C07272=1088.539,208.717,-73.617,176.065,20.904,153.231
C07273=1088.530,208.334,-73.580,176.061,20.901,153.231
C07274=1088.507,207.310,-73.481,175.988,20.864,153.235
C07275=1088.502,207.061,-73.457,175.986,20.863,153.235
C07276=1088.497,206.812,-73.433,175.983,20.861,153.235
C07277=1088.490,206.563,-73.409,175.980,20.859,153.235
C07278=1088.485,206.314,-73.385,175.977,20.858,153.236
C07279=1088.479,206.066,-73.361,175.974,20.857,153.236
C07280=1088.474,205.817,-73.337,175.972,20.855,153.236
C07281=1088.469,205.568,-73.314,175.969,20.854,153.236
C07282=1088.463,205.320,-73.290,175.965,20.852,153.236
C07283=1088.457,205.071,-73.265,175.963,20.851,153.236
C07284=1088.452,204.821,-73.242,175.960,20.850,153.237
C07285=1088.446,204.573,-73.218,175.958,20.848,153.237
C07286=1088.441,204.324,-73.195,175.955,20.847,153.237
C07287=1088.435,204.076,-73.171,175.952,20.845,153.237
C07288=1088.429,203.827,-73.147,175.949,20.844,153.237
C07289=1088.424,203.578,-73.123,175.946,20.842,153.237
C07290=1088.418,203.329,-73.099,175.944,20.841,153.237
C07291=1088.413,203.080,-73.076,175.941,20.839,153.237
C07292=1088.407,202.831,-73.052,175.938,20.838,153.238
C07293=1088.402,202.582,-73.028,175.936,20.837,153.238
C07294=1088.396,202.334,-73.005,175.933,20.836,153.238
C07295=1088.391,202.085,-72.981,175.929,20.834,153.238
C07296=1088.385,201.836,-72.957,175.927,20.833,153.238
C07297=1088.378,201.587,-72.934,175.924,20.831,153.238
C07298=1088.373,201.338,-72.910,175.922,20.830,153.239
C07299=1088.367,201.089,-72.887,175.919,20.829,153.239
C07300=1088.361,200.841,-72.863,175.916,20.827,153.239
C07301=1088.356,200.592,-72.840,175.914,20.826,153.239
C07302=1088.350,200.344,-72.816,175.910,20.824,153.239
C07303=1088.345,200.095,-72.793,175.907,20.823,153.239
C07304=1088.340,199.845,-72.770,175.905,20.822,153.240
C07305=1088.334,199.597,-72.746,175.902,20.820,153.240
C07306=1088.327,199.348,-72.723,175.899,20.819,153.240
C07307=1088.322,199.098,-72.699,175.897,20.818,153.240
C07308=1088.316,198.850,-72.675,175.894,20.816,153.240
C07309=1088.310,198.601,-72.652,175.891,20.814,153.240
C07310=1088.305,198.353,-72.628,175.888,20.813,153.241
C07311=1088.299,198.104,-72.605,175.885,20.812,153.241
C07312=1088.294,197.855,-72.582,175.883,20.811,153.241
C07313=1088.289,197.606,-72.559,175.880,20.809,153.241
C07314=1088.283,197.357,-72.535,175.877,20.808,153.241
C07315=1088.277,197.108,-72.512,175.875,20.807,153.241
C07316=1088.272,196.859,-72.489,175.872,20.805,153.241
C07317=1088.266,196.611,-72.465,175.870,20.804,153.241
C07318=1088.260,196.362,-72.442,175.866,20.802,153.242
C07319=1088.254,196.113,-72.419,175.863,20.801,153.242
C07320=1088.249,195.864,-72.396,175.861,20.800,153.242
C07321=1088.244,195.615,-72.373,175.858,20.798,153.242
C07322=1088.238,195.367,-72.349,175.856,20.797,153.242
C07323=1088.233,195.118,-72.325,175.853,20.795,153.242
C07324=1088.227,194.869,-72.302,175.850,20.794,153.243
C07325=1088.221,194.620,-72.279,175.848,20.793,153.243
C07326=1088.216,194.371,-72.257,175.845,20.791,153.243
C07327=1088.211,194.122,-72.233,175.842,20.790,153.243
C07328=1088.205,193.873,-72.209,175.840,20.788,153.243
C07329=1088.199,193.624,-72.186,175.836,20.787,153.243
C07330=1088.193,193.376,-72.163,175.834,20.786,153.243
C07331=1088.187,193.127,-72.141,175.831,20.784,153.244
C07332=1088.182,192.877,-72.117,175.828,20.783,153.244
C07333=1088.177,192.629,-72.094,175.826,20.781,153.244
C07334=1088.171,192.380,-72.071,175.823,20.780,153.244
C07335=1088.165,192.103,-72.046,175.821,20.778,153.244
C07336=1088.159,191.825,-72.019,175.817,20.777,153.244
C07337=1088.153,191.548,-71.994,175.814,20.775,153.244
C07338=1088.146,191.270,-71.968,175.811,20.774,153.245
C07339=1088.141,191.021,-71.945,175.808,20.772,153.245
C07340=1088.135,190.772,-71.922,175.806,20.771,153.245
C07341=1088.130,190.523,-71.899,175.803,20.769,153.245
C07342=1088.125,190.275,-71.876,175.801,20.768,153.245
C07343=1088.119,190.026,-71.853,175.798,20.766,153.245
C07344=1088.113,189.777,-71.831,175.795,20.765,153.245
C07345=1088.108,189.528,-71.807,175.793,20.763,153.245
C07346=1088.102,189.279,-71.784,175.790,20.762,153.246
C07347=1088.097,189.030,-71.761,175.787,20.761,153.246
C07348=1088.091,188.782,-71.739,175.785,20.760,153.246
C07349=1088.086,188.533,-71.716,175.782,20.758,153.246
C07350=1088.080,188.284,-71.693,175.780,20.757,153.246
C07351=1088.075,188.035,-71.670,175.777,20.755,153.246
C07352=1088.070,187.786,-71.647,175.775,20.754,153.246
C07353=1088.064,187.537,-71.624,175.771,20.752,153.246
C07354=1088.059,187.289,-71.601,175.768,20.750,153.247
C07355=1088.053,187.040,-71.578,175.766,20.749,153.247
C07356=1088.048,186.790,-71.556,175.763,20.748,153.247
C07357=1088.042,186.541,-71.533,175.761,20.746,153.247
C07358=1088.037,186.293,-71.511,175.758,20.745,153.247
C07359=1088.031,186.044,-71.488,175.756,20.743,153.247
C07360=1088.025,185.795,-71.465,175.753,20.742,153.247
C07361=1088.021,185.545,-71.442,175.750,20.740,153.247
C07362=1088.015,185.297,-71.419,175.748,20.739,153.247
C07363=1088.010,185.048,-71.396,175.745,20.737,153.248
C07364=1088.003,184.800,-71.374,175.743,20.736,153.248
C07365=1087.998,184.550,-71.352,175.740,20.735,153.248
C07366=1087.992,184.301,-71.329,175.737,20.734,153.248
C07367=1087.986,184.053,-71.306,175.735,20.732,153.248
C07368=1087.981,183.803,-71.284,175.732,20.731,153.248
C07369=1087.974,183.554,-71.261,175.729,20.729,153.248
C07370=1087.969,183.306,-71.239,175.727,20.728,153.249
C07371=1087.964,183.057,-71.217,175.724,20.727,153.249
C07372=1087.958,182.808,-71.194,175.722,20.725,153.249
C07373=1087.952,182.559,-71.171,175.719,20.724,153.249
C07374=1087.946,182.310,-71.149,175.716,20.722,153.249
C07375=1087.941,182.061,-71.126,175.714,20.722,153.249
C07376=1087.935,181.813,-71.104,175.711,20.720,153.249
C07377=1087.929,181.563,-71.082,175.708,20.719,153.250
C07378=1087.924,181.315,-71.059,175.706,20.717,153.250
C07379=1087.918,181.065,-71.037,175.703,20.716,153.250
C07380=1087.912,180.816,-71.014,175.701,20.714,153.250
C07381=1087.907,180.568,-70.992,175.698,20.713,153.250
C07382=1087.901,180.319,-70.969,175.695,20.712,153.250
C07383=1087.895,180.070,-70.947,175.693,20.710,153.250
C07384=1087.889,179.821,-70.925,175.690,20.709,153.251
C07385=1087.884,179.572,-70.902,175.687,20.708,153.251
C07386=1087.878,179.323,-70.881,175.685,20.706,153.251
C07387=1087.872,179.074,-70.858,175.682,20.705,153.251
C07388=1087.867,178.825,-70.836,175.680,20.703,153.251
C07389=1087.861,178.576,-70.814,175.677,20.702,153.251
C07390=1087.855,178.327,-70.791,175.675,20.700,153.251
C07391=1087.850,178.078,-70.769,175.672,20.699,153.252
C07392=1087.844,177.829,-70.747,175.669,20.698,153.252
C07393=1087.839,177.580,-70.725,175.667,20.696,153.252
C07394=1087.833,177.332,-70.702,175.664,20.695,153.252
C07395=1087.827,177.082,-70.680,175.661,20.694,153.252
C07396=1087.822,176.834,-70.658,175.659,20.692,153.252
C07397=1087.816,176.585,-70.635,175.656,20.691,153.252
C07398=1087.810,176.335,-70.614,175.654,20.689,153.252
C07399=1087.804,176.058,-70.589,175.651,20.688,153.252
C07400=1087.798,175.780,-70.564,175.648,20.686,153.253
C07401=1087.792,175.502,-70.539,175.645,20.684,153.253
C07402=1087.785,175.225,-70.515,175.642,20.683,153.253
C07403=1087.780,174.976,-70.493,175.640,20.682,153.253
C07404=1087.774,174.727,-70.471,175.637,20.680,153.253
C07405=1087.768,174.477,-70.449,175.635,20.679,153.253
C07406=1087.763,174.229,-70.426,175.632,20.677,153.253
C07407=1087.757,173.980,-70.405,175.630,20.676,153.253
C07408=1087.752,173.731,-70.383,175.627,20.674,153.254
C07409=1087.746,173.482,-70.361,175.624,20.673,153.254
C07410=1087.740,173.233,-70.338,175.623,20.672,153.254
C07411=1087.736,172.984,-70.316,175.620,20.670,153.254
C07412=1087.729,172.735,-70.295,175.617,20.669,153.254
C07413=1087.724,172.486,-70.272,175.615,20.668,153.254
C07414=1087.718,172.238,-70.250,175.612,20.666,153.254
C07415=1087.713,171.988,-70.228,175.610,20.665,153.254
C07416=1087.707,171.740,-70.207,175.607,20.663,153.254
C07417=1087.702,171.490,-70.185,175.605,20.662,153.255
C07418=1087.696,171.242,-70.163,175.602,20.660,153.255
C07419=1087.691,170.992,-70.141,175.600,20.658,153.255
C07420=1087.685,170.743,-70.119,175.597,20.657,153.255
C07421=1087.679,170.495,-70.097,175.594,20.655,153.255
C07422=1087.674,170.245,-70.075,175.592,20.654,153.255
C07423=1087.668,169.997,-70.053,175.589,20.653,153.255
C07424=1087.663,169.747,-70.031,175.587,20.651,153.255
C07425=1087.657,169.499,-70.010,175.584,20.650,153.255
C07426=1087.652,169.249,-69.988,175.582,20.649,153.255
C07427=1087.646,169.001,-69.966,175.580,20.647,153.256
C07428=1087.641,168.751,-69.944,175.577,20.645,153.256
C07429=1087.635,168.503,-69.923,175.575,20.644,153.256
C07430=1087.630,168.253,-69.901,175.572,20.642,153.256
C07431=1087.624,168.005,-69.879,175.570,20.641,153.256
C07432=1087.619,167.755,-69.857,175.567,20.640,153.256
C07433=1087.613,167.507,-69.836,175.564,20.638,153.256
C07434=1087.608,167.257,-69.814,175.562,20.637,153.256
C07435=1087.603,167.009,-69.792,175.560,20.635,153.256
C07436=1087.597,166.759,-69.770,175.557,20.633,153.256
C07437=1087.592,166.511,-69.749,175.554,20.632,153.257
C07438=1087.587,166.262,-69.727,175.553,20.631,153.257
C07439=1087.581,166.012,-69.705,175.550,20.629,153.257
C07440=1087.575,165.764,-69.684,175.548,20.627,153.257
C07441=1087.570,165.514,-69.662,175.545,20.626,153.257
C07442=1087.564,165.266,-69.641,175.543,20.625,153.257
C07443=1087.559,165.016,-69.618,175.540,20.623,153.257
C07444=1087.553,164.767,-69.598,175.537,20.622,153.257
C07445=1087.548,164.519,-69.576,175.535,20.620,153.257
C07446=1087.542,164.269,-69.554,175.532,20.618,153.257
C07447=1087.537,164.021,-69.533,175.530,20.617,153.257
C07448=1087.531,163.771,-69.511,175.528,20.616,153.257
C07449=1087.526,163.523,-69.490,175.526,20.614,153.257
C07450=1087.521,163.274,-69.468,175.523,20.613,153.258
C07451=1087.515,163.024,-69.447,175.521,20.611,153.258
C07452=1087.510,162.775,-69.425,175.518,20.610,153.258
C07453=1087.505,162.527,-69.404,175.516,20.608,153.258
C07454=1087.499,162.278,-69.382,175.513,20.606,153.258
C07455=1087.494,162.028,-69.361,175.510,20.605,153.258
C07456=1087.488,161.779,-69.339,175.509,20.603,153.258
C07457=1087.482,161.530,-69.318,175.506,20.602,153.258
C07458=1087.477,161.282,-69.296,175.504,20.600,153.258
C07459=1087.472,161.032,-69.275,175.501,20.599,153.258
C07460=1087.466,160.783,-69.254,175.499,20.598,153.258
C07461=1087.460,160.534,-69.232,175.496,20.596,153.258
C07462=1087.454,160.286,-69.211,175.494,20.594,153.259
C07463=1087.449,160.007,-69.187,175.491,20.593,153.259
C07464=1087.442,159.729,-69.164,175.489,20.591,153.259
C07465=1087.436,159.451,-69.140,175.486,20.590,153.259
C07466=1087.429,159.173,-69.117,175.483,20.588,153.259
C07467=1087.424,158.924,-69.095,175.481,20.586,153.259
C07468=1087.419,158.675,-69.074,175.478,20.585,153.259
C07469=1087.413,158.425,-69.052,175.476,20.584,153.259
C07470=1087.407,158.177,-69.031,175.473,20.582,153.259
C07471=1087.402,157.928,-69.011,175.471,20.580,153.259
C07472=1087.396,157.679,-68.989,175.468,20.579,153.260
C07473=1087.390,157.430,-68.968,175.467,20.578,153.260
C07474=1087.385,157.181,-68.947,175.464,20.576,153.260
C07475=1087.379,156.932,-68.926,175.461,20.575,153.260
C07476=1087.374,156.683,-68.905,175.459,20.573,153.260
C07477=1087.368,156.434,-68.884,175.456,20.571,153.260
C07478=1087.363,156.184,-68.862,175.454,20.570,153.260
C07479=1087.357,155.936,-68.841,175.452,20.568,153.260
C07480=1087.352,155.686,-68.820,175.450,20.567,153.260
C07481=1087.346,155.437,-68.799,175.447,20.566,153.260
C07482=1087.341,155.188,-68.778,175.445,20.564,153.260
C07483=1087.335,154.940,-68.757,175.442,20.562,153.260
C07484=1087.329,154.690,-68.736,175.440,20.561,153.260
C07485=1087.324,154.441,-68.715,175.437,20.559,153.261
C07486=1087.318,154.192,-68.694,175.435,20.558,153.261
C07487=1087.312,153.943,-68.673,175.433,20.556,153.261
C07488=1087.306,153.694,-68.653,175.430,20.555,153.261
C07489=1087.301,153.445,-68.632,175.428,20.554,153.261
C07490=1087.295,153.196,-68.610,175.425,20.552,153.261
C07491=1087.290,152.947,-68.590,175.423,20.550,153.261
C07492=1087.284,152.698,-68.569,175.421,20.549,153.261
C07493=1087.279,152.449,-68.548,175.419,20.548,153.261
C07494=1087.273,152.199,-68.527,175.416,20.546,153.261
C07495=1087.267,151.951,-68.506,175.414,20.544,153.261
C07496=1087.262,151.702,-68.485,175.411,20.543,153.261
C07497=1087.257,151.452,-68.465,175.410,20.541,153.261
C07498=1087.251,151.203,-68.443,175.407,20.540,153.262
C07499=1087.245,150.954,-68.423,175.404,20.539,153.262
C07500=1087.240,150.705,-68.402,175.402,20.537,153.262
C07501=1087.235,150.456,-68.381,175.399,20.535,153.262
C07502=1087.228,150.207,-68.360,175.397,20.534,153.262
C07503=1087.223,149.958,-68.340,175.395,20.532,153.262
C07504=1087.217,149.709,-68.319,175.393,20.531,153.262
C07505=1087.212,149.460,-68.298,175.390,20.529,153.262
C07506=1087.206,149.210,-68.277,175.388,20.527,153.262
C07507=1087.201,148.961,-68.257,175.385,20.526,153.262
C07508=1087.195,148.713,-68.235,175.384,20.525,153.262
C07509=1087.189,148.464,-68.215,175.381,20.523,153.262
C07510=1087.184,148.215,-68.195,175.379,20.522,153.262
C07511=1087.178,147.965,-68.174,175.376,20.520,153.262
C07512=1087.173,147.716,-68.153,175.374,20.518,153.262
C07513=1087.167,147.468,-68.133,175.372,20.517,153.263
C07514=1087.161,147.219,-68.112,175.369,20.516,153.263
C07515=1087.156,146.969,-68.091,175.367,20.514,153.263
C07516=1087.150,146.720,-68.071,175.364,20.512,153.263
C07517=1087.144,146.471,-68.051,175.362,20.511,153.263
C07518=1087.139,146.222,-68.030,175.360,20.509,153.263
C07519=1087.134,145.973,-68.010,175.358,20.508,153.263
C07520=1087.127,145.724,-67.989,175.355,20.506,153.263
C07521=1087.122,145.475,-67.968,175.353,20.505,153.263
C07522=1087.116,145.225,-67.947,175.351,20.504,153.263
C07523=1087.111,144.976,-67.927,175.349,20.502,153.263
C07524=1087.105,144.727,-67.907,175.346,20.500,153.263
C07525=1087.100,144.478,-67.886,175.344,20.498,153.263
C07526=1087.094,144.229,-67.865,175.341,20.497,153.263
C07527=1087.087,143.951,-67.843,175.339,20.495,153.264
C07528=1087.081,143.672,-67.820,175.336,20.493,153.264
C07529=1087.075,143.394,-67.797,175.334,20.492,153.264
C07530=1087.069,143.116,-67.774,175.331,20.490,153.264
C07531=1087.064,142.867,-67.754,175.329,20.489,153.264
C07532=1087.057,142.618,-67.733,175.327,20.487,153.264
C07533=1087.052,142.368,-67.714,175.325,20.486,153.264
C07534=1087.047,142.119,-67.693,175.322,20.484,153.264
C07535=1087.041,141.870,-67.673,175.320,20.482,153.264
C07536=1087.036,141.621,-67.652,175.317,20.480,153.264
C07537=1087.030,141.372,-67.632,175.316,20.479,153.264
C07538=1087.025,141.123,-67.612,175.313,20.477,153.264
C07539=1087.019,140.874,-67.591,175.311,20.476,153.264
C07540=1087.013,140.625,-67.571,175.308,20.474,153.264
C07541=1087.008,140.376,-67.551,175.307,20.473,153.264
C07542=1087.001,140.126,-67.531,175.304,20.471,153.264
C07543=1086.996,139.877,-67.510,175.302,20.470,153.264
C07544=1086.990,139.628,-67.490,175.299,20.468,153.264
C07545=1086.985,139.379,-67.470,175.298,20.467,153.264
C07546=1086.980,139.129,-67.450,175.295,20.465,153.264
C07547=1086.974,138.881,-67.430,175.293,20.463,153.264
C07548=1086.969,138.632,-67.409,175.290,20.461,153.264
C07549=1086.963,138.383,-67.389,175.289,20.460,153.265
C07550=1086.957,138.134,-67.369,175.286,20.459,153.265
C07551=1086.952,137.884,-67.349,175.284,20.457,153.265
C07552=1086.946,137.635,-67.329,175.281,20.455,153.265
C07553=1086.941,137.386,-67.309,175.280,20.454,153.265
C07554=1086.935,137.137,-67.289,175.277,20.452,153.265
C07555=1086.929,136.888,-67.268,175.275,20.451,153.265
C07556=1086.924,136.639,-67.249,175.272,20.449,153.265
C07557=1086.918,136.389,-67.228,175.271,20.448,153.265
C07558=1086.912,136.140,-67.208,175.268,20.446,153.265
C07559=1086.906,135.891,-67.188,175.266,20.444,153.265
C07560=1086.901,135.642,-67.168,175.264,20.443,153.265
C07561=1086.895,135.393,-67.148,175.262,20.442,153.265
C07562=1086.890,135.144,-67.128,175.259,20.440,153.265
C07563=1086.884,134.894,-67.109,175.257,20.438,153.265
C07564=1086.879,134.645,-67.088,175.255,20.437,153.265
C07565=1086.873,134.396,-67.068,175.253,20.435,153.265
C07566=1086.867,134.147,-67.049,175.250,20.433,153.265
C07567=1086.862,133.898,-67.028,175.248,20.431,153.265
C07568=1086.856,133.649,-67.008,175.246,20.430,153.265
C07569=1086.851,133.399,-66.989,175.244,20.428,153.265
C07570=1086.845,133.150,-66.969,175.241,20.427,153.265
C07571=1086.839,132.902,-66.949,175.240,20.425,153.265
C07572=1086.834,132.653,-66.929,175.237,20.424,153.265
C07573=1086.828,132.404,-66.909,175.235,20.422,153.266
C07574=1086.823,132.154,-66.890,175.232,20.420,153.266
C07575=1086.817,131.905,-66.869,175.231,20.419,153.266
C07576=1086.811,131.656,-66.849,175.228,20.417,153.266
C07577=1086.806,131.407,-66.830,175.226,20.416,153.266
C07578=1086.800,131.158,-66.810,175.224,20.414,153.266
C07579=1086.794,130.909,-66.791,175.222,20.412,153.266
C07580=1086.789,130.660,-66.770,175.219,20.411,153.266
C07581=1086.783,130.410,-66.751,175.217,20.409,153.266
C07582=1086.777,130.161,-66.731,175.215,20.408,153.266
C07583=1086.771,129.912,-66.712,175.213,20.406,153.266
C07584=1086.765,129.663,-66.692,175.210,20.405,153.266
C07585=1086.760,129.414,-66.673,175.209,20.403,153.266
C07586=1086.755,129.165,-66.652,175.206,20.401,153.266
C07587=1086.749,128.915,-66.633,175.204,20.400,153.266
C07588=1086.743,128.666,-66.613,175.202,20.398,153.266
C07589=1086.737,128.417,-66.594,175.200,20.397,153.266
C07590=1086.731,128.167,-66.575,175.197,20.395,153.266
C07591=1086.725,127.889,-66.553,175.195,20.393,153.266
C07592=1086.719,127.611,-66.530,175.192,20.391,153.266
C07593=1086.713,127.332,-66.509,175.190,20.389,153.266
C07594=1086.706,127.054,-66.487,175.188,20.388,153.266
C07595=1086.700,126.805,-66.467,175.185,20.386,153.266
C07596=1086.694,126.556,-66.448,175.184,20.385,153.266
C07597=1086.689,126.306,-66.428,175.181,20.383,153.266
C07598=1086.683,126.057,-66.408,175.179,20.381,153.266
C07599=1086.678,125.808,-66.388,175.177,20.380,153.266
C07600=1086.673,125.559,-66.370,175.175,20.378,153.266
C07601=1086.667,125.310,-66.350,175.172,20.376,153.266
C07602=1086.661,125.061,-66.330,175.171,20.375,153.266
C07603=1086.655,124.811,-66.311,175.168,20.373,153.266
C07604=1086.649,124.563,-66.291,175.166,20.371,153.267
C07605=1086.644,124.313,-66.272,175.164,20.370,153.266
C07606=1086.638,124.064,-66.253,175.162,20.368,153.266
C07607=1086.633,123.815,-66.234,175.160,20.366,153.266
C07608=1086.627,123.566,-66.214,175.158,20.365,153.267
C07609=1086.621,123.317,-66.195,175.156,20.363,153.267
C07610=1086.615,123.067,-66.175,175.153,20.361,153.267
C07611=1086.610,122.818,-66.156,175.152,20.360,153.266
C07612=1086.604,122.569,-66.136,175.149,20.358,153.267
C07613=1086.599,122.320,-66.117,175.147,20.356,153.267
C07614=1086.594,122.071,-66.097,175.145,20.355,153.267
C07615=1086.588,121.821,-66.078,175.143,20.353,153.267
C07616=1086.582,121.572,-66.059,175.140,20.351,153.267
C07617=1086.576,121.323,-66.039,175.139,20.350,153.267
C07618=1086.571,121.074,-66.020,175.137,20.348,153.267
C07619=1086.566,120.825,-66.001,175.134,20.346,153.267
C07620=1086.560,120.575,-65.982,175.133,20.345,153.267
C07621=1086.554,120.326,-65.962,175.130,20.343,153.267
C07622=1086.548,120.076,-65.943,175.128,20.341,153.267
C07623=1086.543,119.828,-65.924,175.126,20.340,153.267
C07624=1086.537,119.579,-65.904,175.124,20.338,153.267
C07625=1086.532,119.329,-65.885,175.122,20.336,153.267
C07626=1086.526,119.080,-65.866,175.120,20.334,153.267
C07627=1086.521,118.831,-65.847,175.118,20.333,153.267
C07628=1086.515,118.582,-65.828,175.115,20.331,153.267
C07629=1086.510,118.332,-65.808,175.114,20.329,153.267
C07630=1086.504,118.084,-65.790,175.111,20.327,153.267
C07631=1086.499,117.834,-65.770,175.109,20.326,153.267
C07632=1086.493,117.585,-65.751,175.107,20.324,153.267
C07633=1086.487,117.335,-65.732,175.105,20.322,153.267
C07634=1086.482,117.087,-65.713,175.103,20.321,153.267
C07635=1086.477,116.837,-65.694,175.101,20.319,153.267
C07636=1086.471,116.588,-65.675,175.099,20.317,153.267
C07637=1086.466,116.339,-65.656,175.097,20.316,153.267
C07638=1086.460,116.090,-65.636,175.095,20.314,153.267
C07639=1086.454,115.840,-65.617,175.092,20.312,153.267
C07640=1086.449,115.592,-65.599,175.091,20.310,153.266
C07641=1086.443,115.342,-65.580,175.089,20.308,153.266
C07642=1086.437,115.093,-65.560,175.086,20.306,153.266
C07643=1086.432,114.844,-65.541,175.085,20.305,153.266
C07644=1086.427,114.595,-65.522,175.082,20.303,153.266
C07645=1086.421,114.345,-65.503,175.080,20.301,153.266
C07646=1086.416,114.097,-65.484,175.079,20.300,153.266
C07647=1086.410,113.846,-65.466,175.076,20.298,153.266
C07648=1086.404,113.597,-65.447,175.075,20.297,153.266
C07649=1086.398,113.348,-65.428,175.072,20.295,153.266
C07650=1086.393,113.099,-65.409,175.070,20.293,153.266
C07651=1086.387,112.850,-65.390,175.068,20.291,153.266
C07652=1086.381,112.601,-65.371,175.066,20.289,153.266
C07653=1086.376,112.352,-65.352,175.064,20.287,153.266
C07654=1086.371,112.102,-65.334,175.062,20.286,153.266
C07655=1086.364,111.824,-65.312,175.060,20.284,153.266
C07656=1086.358,111.545,-65.291,175.057,20.282,153.266
C07657=1086.351,111.267,-65.270,175.055,20.280,153.266
C07658=1086.345,110.988,-65.249,175.053,20.278,153.266
C07659=1086.340,110.739,-65.231,175.050,20.276,153.266
C07660=1086.334,110.490,-65.212,175.049,20.275,153.266
C07661=1086.328,110.241,-65.193,175.046,20.273,153.266
C07662=1086.322,109.992,-65.174,175.045,20.272,153.266
C07663=1086.317,109.742,-65.156,175.042,20.270,153.266
C07664=1086.311,109.493,-65.137,175.040,20.268,153.266
C07665=1086.305,109.244,-65.118,175.039,20.266,153.266
C07666=1086.300,108.995,-65.099,175.036,20.264,153.266
C07667=1086.294,108.745,-65.081,175.035,20.263,153.266
C07668=1086.288,108.496,-65.062,175.032,20.261,153.266
C07669=1086.283,108.247,-65.043,175.030,20.259,153.266
C07670=1086.277,107.998,-65.025,175.029,20.257,153.266
C07671=1086.271,107.748,-65.006,175.026,20.256,153.266
C07672=1086.266,107.499,-64.987,175.025,20.254,153.266
C07673=1086.260,107.250,-64.969,175.022,20.252,153.266
C07674=1086.255,107.001,-64.950,175.020,20.251,153.266
C07675=1086.248,106.751,-64.931,175.018,20.249,153.266
C07676=1086.243,106.502,-64.913,175.016,20.247,153.266
C07677=1086.237,106.253,-64.895,175.014,20.246,153.266
C07678=1086.232,106.004,-64.876,175.012,20.244,153.266
C07679=1086.226,105.754,-64.857,175.010,20.242,153.266
C07680=1086.221,105.506,-64.839,175.008,20.240,153.266
C07681=1086.215,105.256,-64.820,175.006,20.238,153.266
C07682=1086.209,105.007,-64.802,175.005,20.236,153.266
C07683=1086.204,104.757,-64.784,175.002,20.234,153.266
C07684=1086.198,104.508,-64.765,175.000,20.232,153.266
C07685=1086.193,104.259,-64.746,174.998,20.231,153.266
C07686=1086.186,104.010,-64.728,174.996,20.229,153.266
C07687=1086.181,103.761,-64.709,174.995,20.228,153.266
C07688=1086.176,103.511,-64.691,174.992,20.226,153.266
C07689=1086.170,103.262,-64.672,174.990,20.224,153.266
C07690=1086.165,103.012,-64.654,174.988,20.222,153.266
C07691=1086.159,102.764,-64.636,174.986,20.220,153.266
C07692=1086.154,102.514,-64.617,174.985,20.219,153.266
C07693=1086.148,102.265,-64.599,174.982,20.217,153.266
C07694=1086.142,102.015,-64.580,174.981,20.215,153.266
C07695=1086.136,101.767,-64.562,174.978,20.213,153.266
C07696=1086.131,101.517,-64.544,174.976,20.211,153.266
C07697=1086.126,101.268,-64.526,174.975,20.209,153.265
C07698=1086.120,101.018,-64.507,174.972,20.207,153.265
C07699=1086.114,100.769,-64.489,174.971,20.206,153.265
C07700=1086.108,100.520,-64.471,174.969,20.204,153.265
C07701=1086.103,100.270,-64.452,174.966,20.202,153.265
C07702=1086.097,100.021,-64.434,174.965,20.201,153.265
C07703=1086.091,99.772,-64.416,174.962,20.199,153.265
C07704=1086.086,99.523,-64.398,174.961,20.197,153.265
C07705=1086.079,99.274,-64.379,174.959,20.195,153.265
C07706=1086.074,99.025,-64.361,174.957,20.194,153.265
C07707=1086.069,98.775,-64.343,174.955,20.192,153.265
C07708=1086.063,98.526,-64.325,174.953,20.190,153.265
C07709=1086.057,98.276,-64.307,174.951,20.188,153.265
C07710=1086.052,98.027,-64.288,174.949,20.186,153.265
C07711=1086.045,97.778,-64.270,174.947,20.185,153.265
C07712=1086.040,97.529,-64.252,174.945,20.183,153.265
C07713=1086.034,97.280,-64.235,174.943,20.181,153.265
C07714=1086.029,97.030,-64.215,174.941,20.179,153.265
C07715=1086.023,96.781,-64.198,174.940,20.177,153.265
C07716=1086.017,96.532,-64.180,174.937,20.175,153.265
C07717=1086.012,96.282,-64.162,174.935,20.173,153.265
C07718=1086.006,96.033,-64.143,174.933,20.172,153.265
C07719=1086.000,95.755,-64.124,174.931,20.170,153.265
C07720=1085.993,95.477,-64.104,174.929,20.168,153.265
C07721=1085.987,95.198,-64.082,174.927,20.166,153.265
C07722=1085.981,94.919,-64.063,174.925,20.164,153.264
C07723=1085.975,94.671,-64.045,174.923,20.162,153.264
C07724=1085.969,94.421,-64.027,174.921,20.160,153.264
C07725=1085.964,94.172,-64.009,174.919,20.158,153.264
C07726=1085.958,93.922,-63.991,174.917,20.156,153.264
C07727=1085.953,93.673,-63.973,174.915,20.155,153.264
C07728=1085.947,93.425,-63.955,174.913,20.153,153.264
C07729=1085.941,93.175,-63.936,174.912,20.151,153.264
C07730=1085.936,92.925,-63.919,174.909,20.149,153.264
C07731=1085.930,92.676,-63.901,174.908,20.147,153.264
C07732=1085.924,92.427,-63.883,174.906,20.145,153.264
C07733=1085.919,92.177,-63.865,174.903,20.143,153.264
C07734=1085.913,91.928,-63.847,174.902,20.141,153.264
C07735=1085.908,91.679,-63.830,174.900,20.139,153.264
C07736=1085.902,91.430,-63.812,174.898,20.138,153.264
C07737=1085.896,91.180,-63.793,174.896,20.136,153.264
C07738=1085.891,90.931,-63.775,174.895,20.134,153.264
C07739=1085.886,90.682,-63.758,174.892,20.132,153.264
C07740=1085.879,90.432,-63.740,174.891,20.131,153.263
C07741=1085.874,90.183,-63.722,174.888,20.129,153.263
C07742=1085.868,89.933,-63.704,174.887,20.127,153.263
C07743=1085.862,89.684,-63.687,174.885,20.125,153.263
C07744=1085.857,89.435,-63.669,174.883,20.123,153.263
C07745=1085.851,89.186,-63.651,174.881,20.121,153.263
C07746=1085.845,88.937,-63.634,174.879,20.120,153.263
C07747=1085.839,88.687,-63.616,174.877,20.118,153.263
C07748=1085.834,88.438,-63.598,174.875,20.116,153.263
C07749=1085.828,88.189,-63.581,174.873,20.114,153.263
C07750=1085.822,87.939,-63.563,174.871,20.112,153.263
C07751=1085.816,87.690,-63.545,174.870,20.110,153.263
C07752=1085.811,87.441,-63.528,174.867,20.108,153.263
C07753=1085.805,87.191,-63.510,174.866,20.106,153.263
C07754=1085.799,86.942,-63.492,174.864,20.104,153.263
C07755=1085.794,86.693,-63.474,174.862,20.103,153.263
C07756=1085.788,86.443,-63.457,174.860,20.101,153.263
C07757=1085.782,86.194,-63.440,174.859,20.099,153.262
C07758=1085.777,85.945,-63.422,174.856,20.097,153.262
C07759=1085.771,85.695,-63.404,174.855,20.096,153.262
C07760=1085.765,85.446,-63.387,174.852,20.094,153.262
C07761=1085.760,85.197,-63.369,174.851,20.092,153.262
C07762=1085.754,84.948,-63.351,174.849,20.090,153.262
C07763=1085.748,84.698,-63.334,174.847,20.088,153.262
C07764=1085.743,84.449,-63.316,174.845,20.086,153.262
C07765=1085.737,84.199,-63.299,174.844,20.084,153.262
C07766=1085.731,83.950,-63.281,174.841,20.082,153.262
C07767=1085.726,83.701,-63.264,174.840,20.081,153.262
C07768=1085.720,83.452,-63.246,174.838,20.078,153.262
C07769=1085.715,83.203,-63.228,174.836,20.077,153.262
C07770=1085.708,82.952,-63.212,174.834,20.075,153.262
C07771=1085.703,82.703,-63.194,174.833,20.073,153.262
C07772=1085.697,82.454,-63.177,174.830,20.071,153.262
C07773=1085.692,82.205,-63.159,174.829,20.069,153.262
C07774=1085.685,81.956,-63.141,174.827,20.067,153.261
C07775=1085.680,81.706,-63.124,174.825,20.065,153.261
C07776=1085.675,81.457,-63.107,174.823,20.063,153.261
C07777=1085.669,81.208,-63.089,174.822,20.061,153.261
C07778=1085.664,80.959,-63.072,174.819,20.060,153.261
C07779=1085.658,80.708,-63.054,174.818,20.058,153.261
C07780=1085.652,80.459,-63.037,174.816,20.056,153.261
C07781=1085.647,80.210,-63.019,174.814,20.054,153.261
C07782=1085.641,79.961,-63.003,174.812,20.052,153.261
C07783=1085.635,79.683,-62.984,174.810,20.050,153.261
C07784=1085.628,79.405,-62.963,174.808,20.047,153.261
C07785=1085.622,79.126,-62.944,174.806,20.046,153.261
C07786=1085.615,78.848,-62.925,174.804,20.043,153.260
C07787=1085.610,78.598,-62.908,174.802,20.041,153.260
C07788=1085.605,78.349,-62.891,174.801,20.039,153.260
C07789=1085.599,78.099,-62.873,174.798,20.037,153.260
C07790=1085.593,77.850,-62.856,174.797,20.036,153.260
C07791=1085.587,77.601,-62.839,174.795,20.033,153.260
C07792=1085.582,77.352,-62.822,174.793,20.032,153.260
C07793=1085.576,77.102,-62.805,174.791,20.030,153.260
C07794=1085.570,76.853,-62.787,174.790,20.028,153.260
C07795=1085.564,76.603,-62.770,174.787,20.026,153.260
C07796=1085.559,76.354,-62.753,174.786,20.024,153.260
C07797=1085.554,76.105,-62.736,174.784,20.022,153.260
C07798=1085.547,75.856,-62.719,174.782,20.020,153.260
C07799=1085.541,75.606,-62.701,174.781,20.018,153.259
C07800=1085.536,75.356,-62.684,174.779,20.016,153.259
C07801=1085.530,75.108,-62.667,174.777,20.015,153.259
C07802=1085.525,74.858,-62.650,174.775,20.012,153.259
C07803=1085.519,74.609,-62.633,174.773,20.011,153.259
C07804=1085.513,74.360,-62.617,174.771,20.009,153.259
C07805=1085.507,74.110,-62.599,174.770,20.007,153.259
C07806=1085.502,73.860,-62.582,174.767,20.005,153.259
C07807=1085.495,73.612,-62.565,174.766,20.003,153.259
C07808=1085.490,73.362,-62.548,174.764,20.001,153.259
C07809=1085.485,73.113,-62.530,174.763,19.999,153.259
C07810=1085.479,72.864,-62.514,174.760,19.997,153.259
C07811=1085.474,72.614,-62.497,174.759,19.995,153.258
C07812=1085.468,72.365,-62.480,174.757,19.993,153.258
C07813=1085.462,72.115,-62.464,174.755,19.992,153.258
C07814=1085.456,71.866,-62.446,174.753,19.989,153.258
C07815=1085.451,71.616,-62.429,174.752,19.988,153.258
C07816=1085.445,71.367,-62.412,174.750,19.985,153.258
C07817=1085.439,71.118,-62.395,174.748,19.984,153.258
C07818=1085.433,70.868,-62.379,174.747,19.982,153.258
C07819=1085.428,70.619,-62.361,174.744,19.980,153.258
C07820=1085.423,70.370,-62.344,174.743,19.978,153.258
C07821=1085.417,70.120,-62.328,174.741,19.976,153.258
C07822=1085.411,69.871,-62.310,174.740,19.974,153.257
C07823=1085.405,69.622,-62.294,174.737,19.972,153.257
C07824=1085.400,69.372,-62.277,174.736,19.970,153.257
C07825=1085.393,69.123,-62.260,174.734,19.968,153.257
C07826=1085.388,68.873,-62.243,174.732,19.966,153.257
C07827=1085.382,68.624,-62.227,174.730,19.964,153.257
C07828=1085.376,68.375,-62.209,174.729,19.962,153.257
C07829=1085.371,68.125,-62.193,174.727,19.960,153.257
C07830=1085.365,67.876,-62.176,174.725,19.958,153.257
C07831=1085.359,67.627,-62.159,174.724,19.956,153.257
C07832=1085.354,67.377,-62.142,174.721,19.954,153.257
C07833=1085.348,67.128,-62.126,174.720,19.952,153.256
C07834=1085.343,66.878,-62.109,174.718,19.950,153.256
C07835=1085.336,66.630,-62.092,174.717,19.948,153.256
C07836=1085.331,66.380,-62.075,174.714,19.946,153.256
C07837=1085.325,66.131,-62.059,174.713,19.944,153.256
C07838=1085.320,65.881,-62.042,174.711,19.943,153.256
C07839=1085.314,65.632,-62.026,174.709,19.941,153.256
C07840=1085.309,65.383,-62.009,174.708,19.939,153.256
C07841=1085.303,65.133,-61.992,174.706,19.937,153.256
C07842=1085.297,64.884,-61.976,174.704,19.935,153.256
C07843=1085.291,64.634,-61.959,174.702,19.933,153.255
C07844=1085.286,64.385,-61.943,174.701,19.931,153.255
C07845=1085.279,64.135,-61.926,174.699,19.929,153.255
C07846=1085.273,63.886,-61.909,174.697,19.927,153.255
C07847=1085.268,63.608,-61.891,174.695,19.925,153.255
C07848=1085.261,63.329,-61.872,174.693,19.923,153.255
C07849=1085.254,63.051,-61.854,174.691,19.921,153.255
C07850=1085.247,62.772,-61.835,174.689,19.919,153.255
C07851=1085.241,62.523,-61.819,174.688,19.917,153.255
C07852=1085.235,62.274,-61.803,174.686,19.915,153.255
C07853=1085.230,62.024,-61.786,174.684,19.913,153.255
C07854=1085.224,61.775,-61.770,174.682,19.911,153.255
C07855=1085.218,61.525,-61.753,174.681,19.909,153.254
C07856=1085.212,61.276,-61.737,174.678,19.907,153.254
C07857=1085.207,61.026,-61.720,174.677,19.905,153.254
C07858=1085.201,60.777,-61.704,174.676,19.903,153.254
C07859=1085.195,60.528,-61.688,174.674,19.901,153.254
C07860=1085.189,60.278,-61.671,174.672,19.899,153.254
C07861=1085.183,60.029,-61.655,174.670,19.897,153.254
C07862=1085.178,59.779,-61.638,174.669,19.895,153.254
C07863=1085.172,59.531,-61.621,174.666,19.893,153.254
C07864=1085.166,59.281,-61.605,174.665,19.891,153.254
C07865=1085.160,59.031,-61.590,174.664,19.889,153.253
C07866=1085.154,58.782,-61.573,174.661,19.887,153.253
C07867=1085.149,58.532,-61.556,174.660,19.885,153.253
C07868=1085.143,58.283,-61.540,174.658,19.883,153.253
C07869=1085.137,58.034,-61.524,174.657,19.881,153.253
C07870=1085.131,57.784,-61.508,174.654,19.879,153.253
C07871=1085.125,57.535,-61.491,174.653,19.877,153.253
C07872=1085.119,57.286,-61.475,174.651,19.876,153.253
C07873=1085.114,57.036,-61.458,174.649,19.873,153.253
C07874=1085.108,56.786,-61.442,174.648,19.871,153.252
C07875=1085.102,56.537,-61.426,174.646,19.869,153.252
C07876=1085.097,56.289,-61.410,174.645,19.867,153.252
C07877=1085.091,56.039,-61.394,174.642,19.865,153.252
C07878=1085.085,55.790,-61.377,174.641,19.863,153.252
C07879=1085.080,55.540,-61.361,174.639,19.862,153.252
C07880=1085.074,55.290,-61.345,174.637,19.859,153.252
C07881=1085.068,55.041,-61.329,174.636,19.857,153.252
C07882=1085.062,54.791,-61.313,174.634,19.855,153.252
C07883=1085.056,54.542,-61.296,174.633,19.853,153.252
C07884=1085.050,54.293,-61.280,174.631,19.852,153.252
C07885=1085.044,54.043,-61.264,174.629,19.849,153.251
C07886=1085.040,53.794,-61.248,174.628,19.847,153.251
C07887=1085.034,53.545,-61.232,174.625,19.845,153.251
C07888=1085.028,53.295,-61.215,174.624,19.843,153.251
C07889=1085.022,53.046,-61.199,174.623,19.842,153.251
C07890=1085.016,52.796,-61.183,174.621,19.839,153.251
C07891=1085.011,52.546,-61.167,174.619,19.837,153.251
C07892=1085.005,52.297,-61.151,174.617,19.835,153.251
C07893=1084.999,52.049,-61.135,174.616,19.833,153.250
C07894=1084.993,51.799,-61.119,174.614,19.831,153.250
C07895=1084.988,51.549,-61.103,174.612,19.829,153.250
C07896=1084.983,51.300,-61.087,174.611,19.827,153.250
C07897=1084.977,51.050,-61.070,174.609,19.825,153.250
C07898=1084.971,50.802,-61.054,174.607,19.823,153.250
C07899=1084.966,50.552,-61.039,174.605,19.821,153.250
C07900=1084.960,50.302,-61.023,174.604,19.819,153.250
C07901=1084.954,50.053,-61.006,174.603,19.818,153.250
C07902=1084.948,49.803,-60.991,174.600,19.815,153.249
C07903=1084.943,49.554,-60.975,174.599,19.813,153.249
C07904=1084.937,49.305,-60.959,174.597,19.811,153.249
C07905=1084.931,49.055,-60.943,174.596,19.809,153.249
C07906=1084.925,48.806,-60.927,174.594,19.807,153.249
C07907=1084.919,48.556,-60.911,174.592,19.805,153.249
C07908=1084.914,48.307,-60.895,174.591,19.803,153.249
C07909=1084.908,48.058,-60.879,174.589,19.801,153.249
C07910=1084.903,47.808,-60.862,174.587,19.799,153.249
C07911=1084.897,47.530,-60.846,174.585,19.797,153.248
C07912=1084.890,47.251,-60.828,174.584,19.795,153.248
C07913=1084.884,46.972,-60.810,174.582,19.792,153.248
C07914=1084.878,46.694,-60.792,174.580,19.790,153.248
C07915=1084.872,46.444,-60.776,174.578,19.788,153.248
C07916=1084.866,46.194,-60.760,174.577,19.786,153.248
C07917=1084.861,45.945,-60.745,174.575,19.784,153.248
C07918=1084.855,45.696,-60.729,174.574,19.782,153.247
C07919=1084.849,45.446,-60.712,174.572,19.779,153.247
C07920=1084.844,45.196,-60.697,174.570,19.778,153.247
C07921=1084.838,44.948,-60.681,174.569,19.776,153.247
C07922=1084.833,44.698,-60.666,174.567,19.773,153.247
C07923=1084.827,44.449,-60.649,174.565,19.771,153.247
C07924=1084.822,44.199,-60.634,174.564,19.770,153.247
C07925=1084.816,43.950,-60.618,174.562,19.767,153.246
C07926=1084.810,43.700,-60.602,174.561,19.765,153.246
C07927=1084.804,43.451,-60.586,174.559,19.763,153.246
C07928=1084.799,43.201,-60.571,174.557,19.761,153.246
C07929=1084.793,42.951,-60.555,174.556,19.759,153.246
C07930=1084.787,42.702,-60.540,174.554,19.757,153.246
C07931=1084.782,42.453,-60.524,174.552,19.755,153.246
C07932=1084.776,42.204,-60.508,174.550,19.753,153.246
C07933=1084.770,41.954,-60.493,174.549,19.751,153.245
C07934=1084.764,41.704,-60.476,174.547,19.749,153.245
C07935=1084.758,41.455,-60.462,174.545,19.747,153.245
C07936=1084.752,41.206,-60.446,174.544,19.744,153.245
C07937=1084.747,40.956,-60.430,174.543,19.743,153.245
C07938=1084.742,40.707,-60.415,174.541,19.741,153.245
C07939=1084.736,40.458,-60.399,174.539,19.738,153.245
C07940=1084.729,40.208,-60.384,174.538,19.736,153.245
C07941=1084.724,39.959,-60.368,174.536,19.734,153.245
C07942=1084.718,39.709,-60.352,174.535,19.732,153.244
C07943=1084.713,39.459,-60.337,174.532,19.730,153.244
C07944=1084.708,39.210,-60.322,174.531,19.728,153.244
C07945=1084.701,38.961,-60.306,174.530,19.726,153.244
C07946=1084.695,38.711,-60.290,174.528,19.724,153.244
C07947=1084.690,38.462,-60.275,174.526,19.722,153.244
C07948=1084.684,38.212,-60.259,174.525,19.720,153.244
C07949=1084.678,37.963,-60.244,174.523,19.718,153.243
C07950=1084.673,37.713,-60.229,174.522,19.716,153.243
C07951=1084.667,37.464,-60.213,174.520,19.713,153.243
C07952=1084.661,37.214,-60.198,174.518,19.712,153.243
C07953=1084.655,36.965,-60.182,174.517,19.710,153.243
C07954=1084.650,36.715,-60.167,174.515,19.707,153.243
C07955=1084.643,36.466,-60.151,174.513,19.706,153.243
C07956=1084.638,36.217,-60.136,174.512,19.704,153.243
C07957=1084.632,35.967,-60.120,174.510,19.701,153.242
C07958=1084.626,35.717,-60.106,174.508,19.700,153.242
C07959=1084.621,35.469,-60.090,174.507,19.698,153.242
C07960=1084.614,35.219,-60.075,174.505,19.695,153.242
C07961=1084.609,34.969,-60.059,174.504,19.694,153.242
C07962=1084.604,34.720,-60.044,174.502,19.692,153.242
C07963=1084.597,34.471,-60.028,174.500,19.689,153.242
C07964=1084.591,34.221,-60.013,174.499,19.687,153.242
C07965=1084.586,33.972,-59.998,174.498,19.686,153.241
C07966=1084.580,33.722,-59.983,174.496,19.683,153.241
C07967=1084.574,33.473,-59.968,174.494,19.681,153.241
C07968=1084.568,33.223,-59.953,174.492,19.679,153.241
C07969=1084.563,32.974,-59.936,174.491,19.677,153.241
C07970=1084.557,32.725,-59.922,174.489,19.675,153.241
C07971=1084.551,32.475,-59.906,174.487,19.673,153.241
C07972=1084.545,32.226,-59.892,174.486,19.671,153.241
C07973=1084.540,31.976,-59.876,174.485,19.669,153.240
C07974=1084.533,31.726,-59.861,174.483,19.667,153.240
C07975=1084.528,31.447,-59.844,174.481,19.665,153.240
C07976=1084.521,31.169,-59.827,174.479,19.662,153.240
C07977=1084.514,30.890,-59.810,174.478,19.660,153.240
C07978=1084.508,30.612,-59.793,174.476,19.658,153.240
C07979=1084.502,30.362,-59.778,174.475,19.656,153.239
C07980=1084.497,30.113,-59.763,174.472,19.654,153.239
C07981=1084.491,29.863,-59.748,174.471,19.652,153.239
C07982=1084.486,29.614,-59.733,174.470,19.650,153.239
C07983=1084.479,29.364,-59.718,174.468,19.647,153.239
C07984=1084.474,29.115,-59.703,174.466,19.646,153.239
C07985=1084.468,28.866,-59.687,174.465,19.644,153.239
C07986=1084.462,28.617,-59.672,174.463,19.641,153.239
C07987=1084.456,28.367,-59.657,174.462,19.639,153.238
C07988=1084.450,28.117,-59.641,174.460,19.638,153.238
C07989=1084.445,27.868,-59.627,174.458,19.635,153.238
C07990=1084.439,27.618,-59.613,174.457,19.633,153.238
C07991=1084.434,27.368,-59.597,174.456,19.631,153.238
C07992=1084.427,27.119,-59.582,174.453,19.629,153.238
C07993=1084.422,26.869,-59.567,174.452,19.627,153.238
C07994=1084.416,26.620,-59.552,174.451,19.625,153.238
C07995=1084.410,26.371,-59.538,174.449,19.623,153.238
C07996=1084.404,26.121,-59.522,174.447,19.621,153.237
C07997=1084.399,25.872,-59.508,174.446,19.619,153.237
C07998=1084.393,25.622,-59.492,174.444,19.617,153.237
C07999=1084.387,25.373,-59.478,174.443,19.615,153.237
C08000=1084.381,25.123,-59.463,174.441,19.613,153.237
C08001=1084.376,24.874,-59.447,174.439,19.611,153.237
C08002=1084.369,24.624,-59.432,174.438,19.609,153.236
C08003=1084.364,24.375,-59.419,174.437,19.607,153.236
C08004=1084.358,24.125,-59.403,174.435,19.605,153.236
C08005=1084.352,23.876,-59.388,174.433,19.603,153.236
C08006=1084.346,23.626,-59.374,174.432,19.601,153.236
C08007=1084.341,23.377,-59.358,174.430,19.599,153.236
C08008=1084.335,23.127,-59.343,174.429,19.597,153.236
C08009=1084.329,22.878,-59.329,174.427,19.595,153.236
C08010=1084.323,22.628,-59.314,174.425,19.592,153.235
C08011=1084.318,22.379,-59.299,174.424,19.591,153.235
C08012=1084.311,22.129,-59.284,174.422,19.588,153.235
C08013=1084.305,21.880,-59.270,174.421,19.586,153.235
C08014=1084.300,21.630,-59.254,174.419,19.584,153.235
C08015=1084.294,21.381,-59.240,174.418,19.582,153.235
C08016=1084.288,21.131,-59.226,174.416,19.580,153.235
C08017=1084.283,20.882,-59.210,174.414,19.578,153.235
C08018=1084.277,20.633,-59.196,174.413,19.576,153.234
C08019=1084.271,20.383,-59.182,174.412,19.574,153.234
C08020=1084.265,20.134,-59.167,174.410,19.572,153.234
C08021=1084.260,19.884,-59.151,174.408,19.570,153.234
C08022=1084.254,19.635,-59.137,174.407,19.568,153.234
C08023=1084.248,19.384,-59.123,174.405,19.565,153.234
C08024=1084.242,19.135,-59.108,174.404,19.564,153.234
C08025=1084.236,18.886,-59.093,174.402,19.562,153.233
C08026=1084.231,18.636,-59.079,174.401,19.560,153.233
C08027=1084.225,18.387,-59.064,174.399,19.557,153.233
C08028=1084.219,18.137,-59.049,174.398,19.556,153.233
C08029=1084.213,17.888,-59.035,174.396,19.554,153.233
C08030=1084.207,17.638,-59.020,174.394,19.551,153.233
C08031=1084.202,17.389,-59.005,174.393,19.549,153.233
C08032=1084.196,17.139,-58.991,174.392,19.548,153.233
C08033=1084.190,16.890,-58.976,174.389,19.545,153.232
C08034=1084.184,16.641,-58.962,174.388,19.543,153.232
C08035=1084.178,16.390,-58.947,174.387,19.541,153.232
C08036=1084.172,16.141,-58.933,174.386,19.539,153.232
C08037=1084.167,15.891,-58.917,174.383,19.537,153.232
C08038=1084.161,15.642,-58.904,174.382,19.535,153.232
C08039=1084.154,15.365,-58.887,174.380,19.533,153.232
C08040=1084.148,15.088,-58.872,174.379,19.531,153.231
C08041=1084.142,14.811,-58.855,174.377,19.528,153.231
C08042=1084.135,14.533,-58.840,174.376,19.526,153.231
C08043=1084.130,14.284,-58.825,174.374,19.524,153.231
C08044=1084.123,14.035,-58.810,174.372,19.522,153.231
C08045=1084.118,13.785,-58.796,174.371,19.520,153.231
C08046=1084.111,13.535,-58.781,174.370,19.518,153.231
C08047=1084.106,13.286,-58.767,174.368,19.516,153.230
C08048=1084.100,13.036,-58.752,174.366,19.514,153.230
C08049=1084.094,12.787,-58.739,174.365,19.512,153.230
C08050=1084.088,12.538,-58.724,174.363,19.509,153.230
C08051=1084.082,12.287,-58.710,174.361,19.508,153.230
C08052=1084.076,12.038,-58.695,174.360,19.506,153.230
C08053=1084.071,11.789,-58.681,174.359,19.504,153.230
C08054=1084.065,11.539,-58.666,174.357,19.501,153.230
C08055=1084.059,11.290,-58.653,174.355,19.500,153.229
C08056=1084.053,11.040,-58.638,174.354,19.498,153.229
C08057=1084.047,10.790,-58.624,174.352,19.495,153.229
C08058=1084.041,10.541,-58.609,174.351,19.494,153.229
C08059=1084.035,10.291,-58.595,174.349,19.492,153.229
C08060=1084.029,10.042,-58.582,174.348,19.490,153.229
C08061=1084.023,9.793,-58.567,174.346,19.487,153.229
C08062=1084.017,9.543,-58.553,174.345,19.486,153.229
C08063=1084.011,9.294,-58.538,174.343,19.484,153.228
C08064=1084.006,9.044,-58.524,174.341,19.481,153.228
C08065=1084.000,8.794,-58.509,174.340,19.479,153.228
C08066=1083.994,8.545,-58.496,174.339,19.478,153.228
C08067=1083.989,8.295,-58.482,174.337,19.476,153.228
C08068=1083.982,8.046,-58.467,174.335,19.473,153.228
C08069=1083.977,7.796,-58.453,174.334,19.472,153.228
C08070=1083.971,7.546,-58.439,174.333,19.470,153.228
C08071=1083.964,7.297,-58.425,174.331,19.468,153.227
C08072=1083.959,7.047,-58.411,174.329,19.465,153.227
C08073=1083.953,6.798,-58.397,174.328,19.464,153.227
C08074=1083.947,6.549,-58.382,174.327,19.462,153.227
C08075=1083.941,6.299,-58.368,174.324,19.459,153.227
C08076=1083.936,6.049,-58.354,174.323,19.457,153.227
C08077=1083.930,5.800,-58.340,174.322,19.456,153.227
C08078=1083.925,5.551,-58.326,174.321,19.453,153.226
C08079=1083.918,5.301,-58.312,174.319,19.451,153.226
C08080=1083.912,5.052,-58.298,174.317,19.449,153.226
C08081=1083.907,4.802,-58.284,174.316,19.447,153.226
C08082=1083.901,4.553,-58.270,174.315,19.445,153.226
C08083=1083.895,4.302,-58.256,174.313,19.443,153.226
C08084=1083.889,4.053,-58.241,174.311,19.441,153.226
C08085=1083.884,3.804,-58.227,174.310,19.439,153.225
C08086=1083.878,3.554,-58.214,174.309,19.437,153.225
C08087=1083.872,3.304,-58.200,174.307,19.435,153.225
C08088=1083.866,3.055,-58.185,174.305,19.433,153.225
C08089=1083.860,2.806,-58.171,174.304,19.431,153.225
C08090=1083.855,2.556,-58.157,174.302,19.429,153.225
C08091=1083.849,2.306,-58.144,174.301,19.427,153.225
C08092=1083.843,2.056,-58.129,174.299,19.425,153.225
C08093=1083.837,1.808,-58.115,174.298,19.423,153.224
C08094=1083.831,1.558,-58.101,174.296,19.421,153.224
C08095=1083.826,1.308,-58.088,174.295,19.419,153.224
C08096=1083.820,1.059,-58.074,174.293,19.417,153.224
C08097=1083.814,0.809,-58.059,174.292,19.415,153.224
C08098=1083.808,0.559,-58.046,174.290,19.412,153.224
C08099=1083.803,0.310,-58.032,174.289,19.411,153.224
C08100=1083.797,0.061,-58.018,174.287,19.409,153.223
C08101=1083.791,-0.189,-58.004,174.286,19.407,153.223
C08102=1083.786,-0.438,-57.990,174.284,19.404,153.223
C08103=1083.779,-0.714,-57.975,174.283,19.402,153.223
C08104=1083.773,-0.989,-57.960,174.281,19.399,153.223
C08105=1083.767,-1.265,-57.945,174.280,19.397,153.223
C08106=1083.760,-1.540,-57.929,174.277,19.395,153.223
C08107=1083.754,-1.789,-57.915,174.276,19.393,153.222
C08108=1083.748,-2.038,-57.901,174.275,19.391,153.222
C08109=1083.743,-2.288,-57.888,174.274,19.389,153.222
C08110=1083.737,-2.538,-57.874,174.272,19.387,153.222
C08111=1083.732,-2.787,-57.860,174.270,19.385,153.222
C08112=1083.725,-3.036,-57.847,174.269,19.383,153.222
C08113=1083.720,-3.286,-57.833,174.268,19.381,153.222
C08114=1083.714,-3.536,-57.818,174.266,19.379,153.221
C08115=1083.708,-3.786,-57.805,174.264,19.377,153.221
C08116=1083.702,-4.035,-57.791,174.263,19.375,153.221
C08117=1083.696,-4.284,-57.778,174.262,19.373,153.221
C08118=1083.690,-4.534,-57.764,174.260,19.371,153.221
C08119=1083.685,-4.784,-57.750,174.258,19.369,153.221
C08120=1083.678,-5.034,-57.737,174.257,19.367,153.221
C08121=1083.673,-5.283,-57.723,174.256,19.365,153.221
C08122=1083.666,-5.532,-57.710,174.254,19.364,153.221
C08123=1083.661,-5.782,-57.696,174.252,19.361,153.220
C08124=1083.655,-6.031,-57.682,174.251,19.359,153.220
C08125=1083.649,-6.281,-57.669,174.249,19.358,153.220
C08126=1083.642,-6.531,-57.655,174.248,19.355,153.220
C08127=1083.637,-6.780,-57.641,174.246,19.353,153.220
C08128=1083.631,-7.030,-57.629,174.245,19.351,153.220
C08129=1083.626,-7.280,-57.615,174.243,19.349,153.220
C08130=1083.619,-7.529,-57.601,174.242,19.347,153.219
C08131=1083.614,-7.779,-57.588,174.240,19.345,153.219
C08132=1083.608,-8.028,-57.574,174.239,19.343,153.219
C08133=1083.602,-8.277,-57.560,174.238,19.341,153.219
C08134=1083.596,-8.527,-57.547,174.236,19.340,153.219
C08135=1083.590,-8.777,-57.533,174.234,19.337,153.219
C08136=1083.584,-9.026,-57.520,174.233,19.335,153.219
C08137=1083.579,-9.276,-57.506,174.232,19.333,153.219
C08138=1083.572,-9.526,-57.493,174.230,19.332,153.219
C08139=1083.567,-9.775,-57.479,174.229,19.330,153.218
C08140=1083.561,-10.025,-57.466,174.227,19.327,153.218
C08141=1083.555,-10.274,-57.452,174.225,19.326,153.218
C08142=1083.549,-10.523,-57.439,174.224,19.324,153.218
C08143=1083.544,-10.774,-57.426,174.223,19.322,153.218
C08144=1083.538,-11.023,-57.413,174.221,19.320,153.218
C08145=1083.532,-11.272,-57.399,174.219,19.318,153.218
C08146=1083.526,-11.522,-57.385,174.218,19.316,153.217
C08147=1083.520,-11.771,-57.372,174.217,19.314,153.217
C08148=1083.514,-12.021,-57.359,174.215,19.312,153.217
C08149=1083.509,-12.271,-57.345,174.213,19.309,153.217
C08150=1083.503,-12.520,-57.332,174.212,19.307,153.217
C08151=1083.497,-12.770,-57.318,174.211,19.306,153.217
C08152=1083.491,-13.020,-57.305,174.210,19.304,153.217
C08153=1083.485,-13.269,-57.292,174.207,19.301,153.217
C08154=1083.479,-13.519,-57.278,174.206,19.300,153.217
C08155=1083.473,-13.769,-57.265,174.205,19.298,153.216
C08156=1083.468,-14.018,-57.251,174.204,19.296,153.216
C08157=1083.462,-14.268,-57.238,174.202,19.294,153.216
C08158=1083.456,-14.517,-57.224,174.200,19.292,153.216
C08159=1083.450,-14.767,-57.212,174.199,19.290,153.216
C08160=1083.444,-15.016,-57.199,174.198,19.288,153.216
C08161=1083.438,-15.266,-57.185,174.196,19.286,153.216
C08162=1083.433,-15.516,-57.172,174.195,19.284,153.215
C08163=1083.426,-15.765,-57.159,174.193,19.282,153.215
C08164=1083.421,-16.015,-57.145,174.191,19.280,153.215
C08165=1083.415,-16.265,-57.132,174.190,19.278,153.215
C08166=1083.409,-16.514,-57.119,174.189,19.277,153.215
C08167=1083.402,-16.787,-57.105,174.187,19.274,153.215
C08168=1083.395,-17.061,-57.091,174.185,19.272,153.215
C08169=1083.390,-17.334,-57.076,174.183,19.269,153.215
C08170=1083.384,-17.608,-57.062,174.182,19.268,153.215
C08171=1083.377,-17.858,-57.049,174.181,19.266,153.214
C08172=1083.371,-18.107,-57.035,174.180,19.264,153.214
C08173=1083.365,-18.357,-57.023,174.177,19.262,153.214
C08174=1083.360,-18.606,-57.009,174.176,19.260,153.214
C08175=1083.354,-18.856,-56.996,174.175,19.258,153.214
C08176=1083.348,-19.105,-56.983,174.173,19.256,153.214
C08177=1083.341,-19.355,-56.970,174.172,19.254,153.214
C08178=1083.336,-19.605,-56.957,174.170,19.252,153.214
C08179=1083.330,-19.854,-56.943,174.169,19.250,153.214
C08180=1083.324,-20.104,-56.931,174.167,19.249,153.213
C08181=1083.318,-20.353,-56.918,174.166,19.247,153.213
C08182=1083.312,-20.603,-56.905,174.165,19.245,153.213
C08183=1083.307,-20.853,-56.891,174.162,19.243,153.213
C08184=1083.301,-21.103,-56.879,174.161,19.241,153.213
C08185=1083.294,-21.352,-56.865,174.160,19.239,153.213
C08186=1083.288,-21.602,-56.853,174.159,19.237,153.213
C08187=1083.283,-21.851,-56.839,174.157,19.235,153.213
C08188=1083.277,-22.101,-56.826,174.155,19.233,153.213
C08189=1083.271,-22.350,-56.813,174.154,19.231,153.212
C08190=1083.266,-22.600,-56.801,174.153,19.229,153.212
C08191=1083.259,-22.849,-56.788,174.151,19.227,153.212
C08192=1083.253,-23.099,-56.775,174.150,19.225,153.212
C08193=1083.248,-23.349,-56.762,174.148,19.223,153.212
C08194=1083.242,-23.598,-56.749,174.146,19.221,153.212
C08195=1083.236,-23.848,-56.736,174.145,19.219,153.212
C08196=1083.230,-24.097,-56.723,174.144,19.218,153.212
C08197=1083.224,-24.347,-56.710,174.142,19.216,153.211
C08198=1083.218,-24.597,-56.697,174.141,19.214,153.211
C08199=1083.213,-24.847,-56.684,174.139,19.212,153.211
C08200=1083.207,-25.096,-56.672,174.138,19.210,153.211
C08201=1083.201,-25.345,-56.658,174.136,19.208,153.211
C08202=1083.195,-25.595,-56.646,174.135,19.206,153.211
C08203=1083.189,-25.845,-56.633,174.134,19.205,153.211
C08204=1083.183,-26.094,-56.620,174.132,19.202,153.211
C08205=1083.177,-26.344,-56.608,174.130,19.200,153.211
C08206=1083.172,-26.594,-56.594,174.129,19.198,153.210
C08207=1083.166,-26.843,-56.581,174.128,19.196,153.210
C08208=1083.161,-27.093,-56.569,174.126,19.195,153.210
C08209=1083.155,-27.343,-56.556,174.125,19.193,153.210
C08210=1083.148,-27.592,-56.543,174.123,19.191,153.210
C08211=1083.142,-27.842,-56.531,174.122,19.189,153.210
C08212=1083.137,-28.092,-56.518,174.120,19.187,153.210
C08213=1083.130,-28.341,-56.505,174.119,19.185,153.210
C08214=1083.124,-28.591,-56.492,174.117,19.184,153.210
C08215=1083.119,-28.841,-56.480,174.116,19.182,153.209
C08216=1083.113,-29.089,-56.467,174.114,19.180,153.210
C08217=1083.106,-29.339,-56.455,174.113,19.178,153.209
C08218=1083.100,-29.589,-56.442,174.111,19.176,153.209
C08219=1083.094,-29.839,-56.430,174.110,19.174,153.209
C08220=1083.088,-30.088,-56.416,174.109,19.173,153.209
C08221=1083.082,-30.338,-56.404,174.107,19.171,153.209
C08222=1083.076,-30.588,-56.391,174.105,19.169,153.209
C08223=1083.071,-30.837,-56.379,174.104,19.167,153.209
C08224=1083.065,-31.087,-56.367,174.102,19.165,153.209
C08225=1083.059,-31.336,-56.353,174.101,19.163,153.209
C08226=1083.053,-31.586,-56.341,174.100,19.161,153.208
C08227=1083.047,-31.836,-56.328,174.099,19.159,153.208
C08228=1083.041,-32.086,-56.316,174.096,19.157,153.208
C08229=1083.036,-32.335,-56.303,174.095,19.155,153.208
C08230=1083.030,-32.584,-56.290,174.094,19.154,153.208
C08231=1083.023,-32.857,-56.277,174.092,19.152,153.208
C08232=1083.017,-33.130,-56.263,174.090,19.149,153.208
C08233=1083.010,-33.402,-56.249,174.089,19.148,153.208
C08234=1083.004,-33.675,-56.236,174.088,19.146,153.208
C08235=1082.998,-33.925,-56.223,174.085,19.144,153.208
C08236=1082.992,-34.175,-56.211,174.084,19.142,153.207
C08237=1082.985,-34.424,-56.198,174.083,19.140,153.207
C08238=1082.980,-34.673,-56.186,174.081,19.138,153.207
C08239=1082.974,-34.923,-56.173,174.080,19.137,153.207
C08240=1082.968,-35.173,-56.161,174.079,19.135,153.207
C08241=1082.962,-35.423,-56.148,174.077,19.133,153.207
C08242=1082.957,-35.672,-56.136,174.075,19.130,153.207
C08243=1082.951,-35.922,-56.123,174.074,19.129,153.207
C08244=1082.945,-36.172,-56.111,174.073,19.127,153.207
C08245=1082.939,-36.421,-56.099,174.071,19.125,153.207
C08246=1082.933,-36.671,-56.087,174.070,19.123,153.206
C08247=1082.927,-36.921,-56.074,174.069,19.122,153.206
C08248=1082.921,-37.170,-56.062,174.066,19.119,153.206
C08249=1082.916,-37.420,-56.049,174.065,19.118,153.206
C08250=1082.910,-37.669,-56.037,174.064,19.116,153.206
C08251=1082.904,-37.919,-56.025,174.062,19.114,153.206
C08252=1082.898,-38.169,-56.012,174.061,19.112,153.206
C08253=1082.892,-38.418,-56.000,174.060,19.111,153.206
C08254=1082.886,-38.668,-55.988,174.058,19.109,153.206
C08255=1082.881,-38.918,-55.975,174.056,19.107,153.206
C08256=1082.874,-39.167,-55.963,174.055,19.105,153.206
C08257=1082.869,-39.417,-55.951,174.054,19.103,153.205
C08258=1082.863,-39.666,-55.938,174.052,19.102,153.205
C08259=1082.856,-39.916,-55.926,174.051,19.100,153.205
C08260=1082.850,-40.166,-55.914,174.049,19.098,153.205
C08261=1082.845,-40.415,-55.902,174.048,19.096,153.205
C08262=1082.838,-40.665,-55.890,174.047,19.094,153.205
C08263=1082.832,-40.915,-55.877,174.044,19.092,153.205
C08264=1082.826,-41.164,-55.865,174.043,19.091,153.205
C08265=1082.820,-41.413,-55.853,174.042,19.089,153.205
C08266=1082.814,-41.663,-55.840,174.040,19.087,153.205
C08267=1082.809,-41.913,-55.828,174.039,19.086,153.205
C08268=1082.802,-42.162,-55.816,174.038,19.084,153.205
C08269=1082.797,-42.412,-55.804,174.036,19.082,153.204
C08270=1082.791,-42.662,-55.791,174.035,19.081,153.204
C08271=1082.784,-42.912,-55.780,174.033,19.078,153.204
C08272=1082.779,-43.161,-55.768,174.031,19.077,153.204
C08273=1082.773,-43.411,-55.755,174.030,19.075,153.204
C08274=1082.766,-43.661,-55.743,174.029,19.073,153.204
C08275=1082.761,-43.910,-55.731,174.027,19.072,153.204
C08276=1082.755,-44.160,-55.718,174.026,19.070,153.204
C08277=1082.749,-44.409,-55.706,174.025,19.068,153.204
C08278=1082.744,-44.659,-55.695,174.023,19.066,153.204
C08279=1082.737,-44.909,-55.683,174.021,19.064,153.204
C08280=1082.731,-45.158,-55.671,174.020,19.062,153.204
C08281=1082.726,-45.408,-55.658,174.018,19.061,153.204
C08282=1082.719,-45.657,-55.646,174.017,19.059,153.203
C08283=1082.713,-45.908,-55.635,174.015,19.057,153.203
C08284=1082.708,-46.157,-55.622,174.014,19.056,153.203
C08285=1082.702,-46.406,-55.610,174.013,19.054,153.203
C08286=1082.696,-46.656,-55.598,174.011,19.052,153.203
C08287=1082.690,-46.905,-55.586,174.009,19.050,153.203
C08288=1082.684,-47.156,-55.574,174.008,19.048,153.203
C08289=1082.679,-47.405,-55.562,174.006,19.047,153.203
C08290=1082.672,-47.654,-55.550,174.005,19.045,153.203
C08291=1082.666,-47.904,-55.538,174.004,19.043,153.203
C08292=1082.660,-48.154,-55.527,174.002,19.042,153.203
C08293=1082.654,-48.404,-55.514,174.001,19.040,153.203
C08294=1082.648,-48.653,-55.503,174.000,19.038,153.203
C08295=1082.643,-48.926,-55.489,173.997,19.036,153.203
C08296=1082.635,-49.200,-55.476,173.996,19.034,153.202
C08297=1082.629,-49.473,-55.463,173.995,19.032,153.202
C08298=1082.622,-49.746,-55.450,173.993,19.031,153.202
C08299=1082.617,-49.995,-55.438,173.991,19.028,153.202
C08300=1082.611,-50.245,-55.426,173.990,19.027,153.202
C08301=1082.605,-50.494,-55.414,173.988,19.025,153.202
C08302=1082.599,-50.744,-55.403,173.987,19.023,153.202
C08303=1082.593,-50.994,-55.391,173.986,19.022,153.202
C08304=1082.587,-51.243,-55.379,173.984,19.020,153.202
C08305=1082.581,-51.493,-55.368,173.983,19.019,153.202
C08306=1082.575,-51.743,-55.355,173.981,19.017,153.202
C08307=1082.569,-51.993,-55.344,173.980,19.016,153.202
C08308=1082.562,-52.242,-55.332,173.979,19.014,153.202
C08309=1082.556,-52.492,-55.320,173.976,19.012,153.202
C08310=1082.551,-52.742,-55.309,173.975,19.010,153.202
C08311=1082.544,-52.991,-55.297,173.973,19.009,153.202
C08312=1082.539,-53.240,-55.285,173.972,19.007,153.201
C08313=1082.532,-53.491,-55.273,173.971,19.006,153.201
C08314=1082.526,-53.740,-55.262,173.969,19.004,153.201
C08315=1082.520,-53.990,-55.251,173.968,19.002,153.201
C08316=1082.514,-54.239,-55.238,173.966,19.000,153.201
C08317=1082.508,-54.489,-55.227,173.965,18.999,153.201
C08318=1082.502,-54.739,-55.215,173.964,18.997,153.201
C08319=1082.496,-54.988,-55.203,173.962,18.996,153.201
C08320=1082.490,-55.238,-55.192,173.961,18.994,153.201
C08321=1082.483,-55.487,-55.180,173.959,18.992,153.201
C08322=1082.478,-55.737,-55.169,173.957,18.990,153.201
C08323=1082.472,-55.987,-55.156,173.956,18.989,153.201
C08324=1082.465,-56.237,-55.145,173.954,18.987,153.201
C08325=1082.459,-56.486,-55.134,173.953,18.986,153.201
C08326=1082.454,-56.736,-55.122,173.951,18.984,153.201
C08327=1082.448,-56.985,-55.110,173.950,18.983,153.201
C08328=1082.441,-57.235,-55.099,173.948,18.981,153.201
C08329=1082.435,-57.484,-55.087,173.947,18.979,153.201
C08330=1082.430,-57.735,-55.076,173.946,18.978,153.201
C08331=1082.424,-57.984,-55.064,173.944,18.976,153.200
C08332=1082.417,-58.234,-55.053,173.943,18.975,153.200
C08333=1082.411,-58.483,-55.041,173.941,18.973,153.200
C08334=1082.406,-58.733,-55.029,173.940,18.971,153.200
C08335=1082.399,-58.983,-55.018,173.939,18.970,153.200
C08336=1082.393,-59.232,-55.006,173.936,18.968,153.200
C08337=1082.387,-59.483,-54.995,173.935,18.966,153.200
C08338=1082.381,-59.731,-54.984,173.934,18.964,153.200
C08339=1082.375,-59.982,-54.972,173.932,18.963,153.200
C08340=1082.370,-60.231,-54.961,173.931,18.961,153.200
C08341=1082.363,-60.481,-54.949,173.929,18.960,153.200
C08342=1082.357,-60.730,-54.938,173.928,18.958,153.200
C08343=1082.351,-60.980,-54.925,173.926,18.957,153.200
C08344=1082.345,-61.230,-54.915,173.925,18.955,153.200
C08345=1082.339,-61.480,-54.903,173.924,18.954,153.200
C08346=1082.333,-61.729,-54.892,173.922,18.952,153.200
C08347=1082.327,-61.978,-54.881,173.921,18.951,153.200
C08348=1082.322,-62.229,-54.869,173.919,18.949,153.200
C08349=1082.316,-62.478,-54.857,173.918,18.948,153.200
C08350=1082.309,-62.728,-54.846,173.917,18.946,153.200
C08351=1082.304,-62.977,-54.835,173.915,18.944,153.200
C08352=1082.297,-63.227,-54.823,173.914,18.943,153.200
C08353=1082.292,-63.477,-54.812,173.911,18.940,153.200
C08354=1082.286,-63.727,-54.801,173.910,18.939,153.200
C08355=1082.280,-63.976,-54.789,173.908,18.937,153.200
C08356=1082.273,-64.226,-54.778,173.907,18.936,153.199
C08357=1082.268,-64.476,-54.767,173.906,18.934,153.199
C08358=1082.261,-64.724,-54.755,173.904,18.933,153.199
C08359=1082.256,-65.000,-54.743,173.903,18.931,153.199
C08360=1082.249,-65.274,-54.730,173.901,18.930,153.199
C08361=1082.242,-65.548,-54.718,173.900,18.928,153.199
C08362=1082.235,-65.823,-54.706,173.898,18.926,153.199
C08363=1082.229,-66.072,-54.694,173.896,18.924,153.199
C08364=1082.224,-66.322,-54.683,173.895,18.923,153.199
C08365=1082.218,-66.572,-54.672,173.893,18.921,153.199
C08366=1082.212,-66.822,-54.661,173.892,18.920,153.199
C08367=1082.205,-67.071,-54.649,173.891,18.918,153.199
C08368=1082.200,-67.321,-54.638,173.889,18.917,153.199
C08369=1082.194,-67.570,-54.627,173.888,18.915,153.199
C08370=1082.188,-67.820,-54.616,173.886,18.914,153.199
C08371=1082.183,-68.070,-54.604,173.885,18.912,153.199
C08372=1082.177,-68.320,-54.593,173.883,18.911,153.199
C08373=1082.170,-68.569,-54.581,173.882,18.909,153.199
C08374=1082.164,-68.819,-54.570,173.880,18.907,153.199
C08375=1082.158,-69.069,-54.559,173.879,18.906,153.199
C08376=1082.152,-69.318,-54.548,173.878,18.904,153.199
C08377=1082.147,-69.568,-54.537,173.876,18.903,153.199
C08378=1082.140,-69.818,-54.526,173.875,18.901,153.199
C08379=1082.134,-70.067,-54.515,173.873,18.900,153.199
C08380=1082.129,-70.317,-54.503,173.872,18.898,153.199
C08381=1082.123,-70.567,-54.492,173.870,18.897,153.199
C08382=1082.117,-70.816,-54.481,173.869,18.895,153.199
C08383=1082.111,-71.066,-54.470,173.867,18.894,153.199
C08384=1082.105,-71.316,-54.459,173.866,18.892,153.199
C08385=1082.099,-71.566,-54.448,173.865,18.891,153.198
C08386=1082.094,-71.815,-54.437,173.863,18.889,153.198
C08387=1082.088,-72.065,-54.426,173.862,18.888,153.198
C08388=1082.082,-72.315,-54.415,173.860,18.886,153.198
C08389=1082.076,-72.564,-54.404,173.859,18.885,153.198
C08390=1082.070,-72.813,-54.393,173.857,18.883,153.198
C08391=1082.064,-73.064,-54.381,173.856,18.882,153.198
C08392=1082.058,-73.313,-54.370,173.853,18.880,153.198
C08393=1082.053,-73.563,-54.359,173.852,18.879,153.198
C08394=1082.047,-73.812,-54.348,173.850,18.877,153.198
C08395=1082.041,-74.062,-54.337,173.849,18.875,153.198
C08396=1082.035,-74.312,-54.326,173.848,18.874,153.198
C08397=1082.029,-74.561,-54.315,173.846,18.872,153.198
C08398=1082.022,-74.811,-54.304,173.845,18.871,153.198
C08399=1082.016,-75.061,-54.294,173.843,18.869,153.198
C08400=1082.011,-75.310,-54.283,173.842,18.868,153.198
C08401=1082.004,-75.560,-54.271,173.840,18.867,153.198
C08402=1081.998,-75.810,-54.261,173.839,18.865,153.198
C08403=1081.993,-76.059,-54.250,173.837,18.864,153.198
C08404=1081.986,-76.309,-54.238,173.836,18.862,153.198
C08405=1081.981,-76.559,-54.228,173.834,18.861,153.198
C08406=1081.974,-76.808,-54.217,173.833,18.860,153.198
C08407=1081.968,-77.058,-54.206,173.832,18.859,153.198
C08408=1081.962,-77.308,-54.196,173.831,18.857,153.198
C08409=1081.957,-77.558,-54.185,173.829,18.856,153.198
C08410=1081.951,-77.807,-54.174,173.828,18.854,153.198
C08411=1081.945,-78.058,-54.163,173.826,18.853,153.198
C08412=1081.939,-78.307,-54.152,173.825,18.852,153.198
C08413=1081.932,-78.556,-54.142,173.823,18.850,153.198
C08414=1081.926,-78.806,-54.131,173.822,18.849,153.198
C08415=1081.920,-79.056,-54.120,173.820,18.847,153.198
C08416=1081.915,-79.305,-54.109,173.818,18.846,153.198
C08417=1081.909,-79.555,-54.098,173.817,18.844,153.198
C08418=1081.903,-79.806,-54.087,173.816,18.843,153.198
C08419=1081.896,-80.055,-54.077,173.814,18.841,153.198
C08420=1081.891,-80.304,-54.066,173.812,18.840,153.198
C08421=1081.885,-80.554,-54.055,173.811,18.839,153.198
C08422=1081.878,-80.804,-54.045,173.810,18.837,153.198
C08423=1081.872,-81.080,-54.033,173.808,18.836,153.198
C08424=1081.865,-81.357,-54.021,173.806,18.834,153.198
C08425=1081.857,-81.634,-54.009,173.804,18.833,153.198
C08426=1081.851,-81.910,-53.997,173.803,18.831,153.198
C08427=1081.845,-82.159,-53.987,173.801,18.830,153.198
C08428=1081.839,-82.410,-53.977,173.800,18.829,153.198
C08429=1081.833,-82.660,-53.965,173.798,18.827,153.198
C08430=1081.826,-82.909,-53.955,173.796,18.826,153.198
C08431=1081.821,-83.158,-53.944,173.795,18.825,153.198
C08432=1081.814,-83.409,-53.933,173.794,18.823,153.198
C08433=1081.808,-83.658,-53.923,173.792,18.822,153.198
C08434=1081.802,-83.908,-53.912,173.790,18.821,153.198
C08435=1081.797,-84.157,-53.902,173.789,18.820,153.199
C08436=1081.790,-84.407,-53.891,173.787,18.818,153.199
C08437=1081.784,-84.657,-53.881,173.786,18.817,153.199
C08438=1081.778,-84.907,-53.870,173.785,18.816,153.199
C08439=1081.772,-85.156,-53.860,173.784,18.815,153.199
C08440=1081.766,-85.406,-53.849,173.782,18.813,153.199
C08441=1081.759,-85.656,-53.839,173.780,18.812,153.199
C08442=1081.754,-85.906,-53.828,173.779,18.811,153.199
C08443=1081.748,-86.155,-53.817,173.777,18.810,153.199
C08444=1081.741,-86.404,-53.807,173.776,18.808,153.199
C08445=1081.735,-86.655,-53.796,173.774,18.806,153.199
C08446=1081.729,-86.904,-53.786,173.773,18.805,153.199
C08447=1081.723,-87.154,-53.775,173.771,18.804,153.199
C08448=1081.718,-87.404,-53.765,173.770,18.803,153.199
C08449=1081.711,-87.653,-53.755,173.768,18.801,153.199
C08450=1081.705,-87.903,-53.743,173.766,18.800,153.199
C08451=1081.699,-88.153,-53.734,173.765,18.799,153.199
C08452=1081.693,-88.402,-53.723,173.764,18.797,153.199
C08453=1081.687,-88.652,-53.713,173.762,18.796,153.199
C08454=1081.681,-88.902,-53.703,173.760,18.795,153.199
C08455=1081.675,-89.151,-53.692,173.759,18.794,153.199
C08456=1081.668,-89.401,-53.681,173.758,18.793,153.199
C08457=1081.663,-89.651,-53.671,173.756,18.792,153.199
C08458=1081.656,-89.900,-53.661,173.755,18.790,153.199
C08459=1081.651,-90.151,-53.650,173.754,18.789,153.199
C08460=1081.644,-90.400,-53.640,173.752,18.788,153.199
C08461=1081.639,-90.649,-53.629,173.750,18.786,153.199
C08462=1081.633,-90.900,-53.619,173.749,18.785,153.199
C08463=1081.626,-91.149,-53.608,173.747,18.784,153.199
C08464=1081.621,-91.399,-53.598,173.746,18.783,153.199
C08465=1081.614,-91.648,-53.588,173.744,18.781,153.199
C08466=1081.609,-91.899,-53.578,173.742,18.780,153.199
C08467=1081.602,-92.148,-53.568,173.741,18.779,153.199
C08468=1081.597,-92.398,-53.557,173.739,18.778,153.200
C08469=1081.590,-92.647,-53.547,173.738,18.776,153.199
C08470=1081.584,-92.897,-53.536,173.737,18.776,153.200
C08471=1081.578,-93.147,-53.526,173.736,18.774,153.200
C08472=1081.572,-93.397,-53.515,173.734,18.773,153.200
C08473=1081.567,-93.647,-53.505,173.732,18.772,153.200
C08474=1081.560,-93.896,-53.495,173.731,18.771,153.200
C08475=1081.555,-94.146,-53.485,173.729,18.769,153.200
C08476=1081.548,-94.395,-53.474,173.728,18.768,153.200
C08477=1081.543,-94.645,-53.464,173.726,18.767,153.200
C08478=1081.537,-94.894,-53.454,173.725,18.766,153.200
C08479=1081.531,-95.144,-53.444,173.723,18.764,153.200
C08480=1081.525,-95.394,-53.434,173.721,18.763,153.200
C08481=1081.519,-95.644,-53.423,173.720,18.761,153.200
C08482=1081.512,-95.894,-53.414,173.719,18.761,153.200
C08483=1081.507,-96.144,-53.403,173.717,18.760,153.200
C08484=1081.500,-96.394,-53.393,173.716,18.758,153.200
C08485=1081.495,-96.643,-53.382,173.714,18.757,153.200
C08486=1081.489,-96.893,-53.373,173.713,18.756,153.200
C08487=1081.482,-97.171,-53.362,173.711,18.755,153.200
C08488=1081.475,-97.450,-53.349,173.710,18.753,153.200
C08489=1081.469,-97.729,-53.338,173.708,18.752,153.200
C08490=1081.462,-98.008,-53.328,173.706,18.750,153.200
C08491=1081.456,-98.258,-53.317,173.705,18.750,153.200
C08492=1081.449,-98.508,-53.307,173.703,18.749,153.201
C08493=1081.443,-98.757,-53.297,173.702,18.747,153.201
C08494=1081.438,-99.008,-53.287,173.700,18.746,153.201
C08495=1081.431,-99.257,-53.277,173.698,18.745,153.201
C08496=1081.425,-99.506,-53.267,173.697,18.744,153.201
C08497=1081.419,-99.756,-53.256,173.695,18.743,153.201
C08498=1081.413,-100.006,-53.247,173.694,18.742,153.201
C08499=1081.407,-100.256,-53.237,173.692,18.741,153.201
C08500=1081.400,-100.505,-53.227,173.691,18.740,153.201
C08501=1081.395,-100.755,-53.217,173.690,18.739,153.201
C08502=1081.389,-101.005,-53.207,173.688,18.738,153.201
C08503=1081.382,-101.254,-53.197,173.686,18.736,153.201
C08504=1081.377,-101.504,-53.187,173.685,18.735,153.201
C08505=1081.371,-101.754,-53.177,173.683,18.734,153.201
C08506=1081.364,-102.003,-53.167,173.681,18.733,153.202
C08507=1081.358,-102.253,-53.157,173.680,18.732,153.202
C08508=1081.352,-102.504,-53.147,173.679,18.731,153.202
C08509=1081.346,-102.753,-53.137,173.677,18.730,153.202
C08510=1081.339,-103.003,-53.127,173.676,18.729,153.202
C08511=1081.334,-103.253,-53.117,173.674,18.728,153.202
C08512=1081.328,-103.502,-53.107,173.673,18.727,153.202
C08513=1081.322,-103.752,-53.098,173.671,18.726,153.202
C08514=1081.315,-104.001,-53.087,173.669,18.725,153.202
C08515=1081.310,-104.252,-53.077,173.669,18.724,153.202
C08516=1081.304,-104.501,-53.068,173.667,18.723,153.202
C08517=1081.297,-104.751,-53.058,173.665,18.722,153.202
C08518=1081.291,-105.000,-53.048,173.664,18.721,153.202
C08519=1081.285,-105.250,-53.038,173.662,18.720,153.203
C08520=1081.279,-105.500,-53.028,173.660,18.718,153.203
C08521=1081.273,-105.750,-53.018,173.659,18.717,153.203
C08522=1081.267,-105.999,-53.008,173.657,18.716,153.203
C08523=1081.261,-106.249,-52.999,173.656,18.716,153.203
C08524=1081.255,-106.499,-52.988,173.654,18.715,153.203
C08525=1081.249,-106.749,-52.979,173.653,18.713,153.203
C08526=1081.243,-106.999,-52.969,173.651,18.712,153.203
C08527=1081.237,-107.248,-52.960,173.650,18.711,153.203
C08528=1081.231,-107.497,-52.950,173.648,18.710,153.203
C08529=1081.225,-107.747,-52.940,173.647,18.710,153.203
C08530=1081.219,-107.997,-52.930,173.645,18.709,153.203
C08531=1081.213,-108.247,-52.921,173.644,18.708,153.204
C08532=1081.207,-108.496,-52.911,173.642,18.707,153.204
C08533=1081.201,-108.746,-52.901,173.641,18.705,153.204
C08534=1081.194,-108.996,-52.892,173.639,18.704,153.204
C08535=1081.188,-109.245,-52.882,173.637,18.703,153.204
C08536=1081.182,-109.495,-52.872,173.636,18.703,153.204
C08537=1081.176,-109.745,-52.862,173.635,18.702,153.204
C08538=1081.169,-109.995,-52.853,173.633,18.701,153.204
C08539=1081.163,-110.244,-52.843,173.631,18.700,153.204
C08540=1081.157,-110.494,-52.834,173.630,18.699,153.204
C08541=1081.151,-110.744,-52.824,173.628,18.698,153.205
C08542=1081.145,-110.994,-52.814,173.627,18.697,153.205
C08543=1081.139,-111.244,-52.804,173.625,18.696,153.205
C08544=1081.133,-111.494,-52.795,173.624,18.695,153.205
C08545=1081.127,-111.744,-52.785,173.622,18.694,153.205
C08546=1081.120,-111.993,-52.775,173.620,18.693,153.205
C08547=1081.114,-112.242,-52.765,173.619,18.693,153.205
C08548=1081.108,-112.492,-52.756,173.618,18.692,153.205
C08549=1081.102,-112.742,-52.746,173.616,18.691,153.205
C08550=1081.096,-112.992,-52.737,173.614,18.690,153.205
C08551=1081.089,-113.268,-52.727,173.613,18.689,153.206
C08552=1081.083,-113.543,-52.716,173.611,18.687,153.206
C08553=1081.076,-113.819,-52.705,173.610,18.686,153.206
C08554=1081.069,-114.094,-52.695,173.608,18.685,153.206
C08555=1081.063,-114.344,-52.686,173.606,18.684,153.206
C08556=1081.057,-114.594,-52.676,173.604,18.684,153.206
C08557=1081.051,-114.844,-52.667,173.603,18.683,153.206
C08558=1081.044,-115.094,-52.657,173.602,18.682,153.206
C08559=1081.039,-115.343,-52.648,173.600,18.681,153.206
C08560=1081.033,-115.593,-52.638,173.598,18.680,153.207
C08561=1081.026,-115.842,-52.629,173.597,18.679,153.207
C08562=1081.020,-116.092,-52.619,173.596,18.679,153.207
C08563=1081.014,-116.342,-52.610,173.594,18.678,153.207
C08564=1081.008,-116.592,-52.600,173.592,18.677,153.207
C08565=1081.002,-116.842,-52.590,173.591,18.676,153.207
C08566=1080.996,-117.091,-52.581,173.589,18.675,153.207
C08567=1080.989,-117.341,-52.571,173.588,18.674,153.207
C08568=1080.984,-117.590,-52.562,173.586,18.673,153.207
C08569=1080.978,-117.840,-52.553,173.585,18.673,153.208
C08570=1080.972,-118.090,-52.544,173.583,18.672,153.208
C08571=1080.966,-118.340,-52.534,173.581,18.671,153.208
C08572=1080.959,-118.590,-52.525,173.580,18.670,153.208
C08573=1080.953,-118.840,-52.516,173.579,18.669,153.208
C08574=1080.946,-119.089,-52.506,173.577,18.668,153.208
C08575=1080.940,-119.339,-52.496,173.575,18.667,153.208
C08576=1080.935,-119.588,-52.487,173.574,18.666,153.208
C08577=1080.928,-119.838,-52.478,173.572,18.666,153.209
C08578=1080.923,-120.088,-52.469,173.571,18.665,153.209
C08579=1080.916,-120.338,-52.459,173.569,18.664,153.209
C08580=1080.910,-120.588,-52.450,173.567,18.663,153.209
C08581=1080.903,-120.838,-52.441,173.566,18.662,153.209
C08582=1080.897,-121.087,-52.431,173.565,18.662,153.209
C08583=1080.892,-121.336,-52.422,173.563,18.661,153.209
C08584=1080.886,-121.587,-52.413,173.561,18.660,153.210
C08585=1080.880,-121.837,-52.404,173.559,18.659,153.210
C08586=1080.873,-122.086,-52.394,173.559,18.659,153.210
C08587=1080.867,-122.336,-52.384,173.557,18.658,153.210
C08588=1080.860,-122.586,-52.375,173.555,18.657,153.210
C08589=1080.855,-122.835,-52.367,173.553,18.656,153.210
C08590=1080.849,-123.085,-52.357,173.552,18.656,153.210
C08591=1080.843,-123.335,-52.348,173.551,18.655,153.210
C08592=1080.837,-123.585,-52.338,173.549,18.654,153.211
C08593=1080.830,-123.834,-52.329,173.547,18.653,153.211
C08594=1080.824,-124.084,-52.321,173.545,18.652,153.211
C08595=1080.818,-124.334,-52.311,173.545,18.652,153.211
C08596=1080.812,-124.584,-52.302,173.543,18.651,153.211
C08597=1080.806,-124.833,-52.292,173.541,18.650,153.211
C08598=1080.799,-125.084,-52.284,173.539,18.649,153.211
C08599=1080.793,-125.333,-52.274,173.538,18.649,153.212
C08600=1080.787,-125.582,-52.265,173.536,18.648,153.212
C08601=1080.782,-125.833,-52.256,173.535,18.647,153.212
C08602=1080.775,-126.082,-52.247,173.533,18.646,153.212
C08603=1080.769,-126.332,-52.238,173.532,18.646,153.212
C08604=1080.762,-126.582,-52.228,173.530,18.645,153.212
C08605=1080.756,-126.831,-52.220,173.529,18.644,153.213
C08606=1080.750,-127.081,-52.211,173.527,18.644,153.213
C08607=1080.744,-127.331,-52.201,173.526,18.643,153.213
C08608=1080.738,-127.581,-52.192,173.524,18.643,153.213
C08609=1080.731,-127.831,-52.183,173.522,18.642,153.213
C08610=1080.727,-128.081,-52.174,173.521,18.641,153.213
C08611=1080.723,-128.337,-52.164,173.519,18.639,153.213
C08612=1080.724,-128.591,-52.152,173.518,18.636,153.213
C08613=1080.728,-128.845,-52.139,173.518,18.633,153.212
C08614=1080.735,-129.097,-52.125,173.518,18.628,153.211
C08615=1080.336,-129.119,-52.266,173.474,18.749,153.242
C08616=1080.329,-128.867,-52.280,173.474,18.754,153.243
C08617=1080.325,-128.613,-52.293,173.474,18.757,153.243
C08618=1080.324,-128.359,-52.305,173.475,18.760,153.244
C08619=1080.326,-128.103,-52.316,173.476,18.762,153.244
C08620=1080.332,-127.853,-52.324,173.478,18.763,153.244
C08621=1080.338,-127.603,-52.334,173.480,18.764,153.244
C08622=1080.344,-127.353,-52.343,173.482,18.764,153.243
C08623=1080.350,-127.103,-52.352,173.483,18.765,153.243
C08624=1080.357,-126.854,-52.361,173.484,18.766,153.243
C08625=1080.363,-126.604,-52.370,173.486,18.766,153.243
C08626=1080.369,-126.354,-52.379,173.488,18.767,153.243
C08627=1080.376,-126.104,-52.388,173.489,18.768,153.243
C08628=1080.382,-125.855,-52.398,173.491,18.769,153.243
C08629=1080.387,-125.605,-52.406,173.492,18.769,153.242
C08630=1080.393,-125.355,-52.416,173.494,18.770,153.242
C08631=1080.400,-125.106,-52.425,173.495,18.771,153.242
C08632=1080.406,-124.855,-52.434,173.497,18.771,153.242
C08633=1080.412,-124.605,-52.443,173.499,18.772,153.242
C08634=1080.418,-124.356,-52.453,173.500,18.773,153.242
C08635=1080.425,-124.107,-52.462,173.501,18.774,153.242
C08636=1080.431,-123.856,-52.470,173.503,18.774,153.241
C08637=1080.437,-123.607,-52.480,173.505,18.775,153.241
C08638=1080.443,-123.357,-52.490,173.507,18.776,153.241
C08639=1080.449,-123.107,-52.499,173.508,18.777,153.241
C08640=1080.455,-122.858,-52.508,173.509,18.778,153.241
C08641=1080.461,-122.608,-52.517,173.511,18.778,153.241
C08642=1080.467,-122.358,-52.526,173.513,18.779,153.240
C08643=1080.474,-122.108,-52.536,173.514,18.780,153.240
C08644=1080.480,-121.858,-52.545,173.515,18.781,153.240
C08645=1080.485,-121.609,-52.554,173.517,18.782,153.240
C08646=1080.491,-121.359,-52.563,173.519,18.782,153.240
C08647=1080.498,-121.109,-52.572,173.521,18.783,153.240
C08648=1080.504,-120.860,-52.582,173.522,18.784,153.240
C08649=1080.510,-120.610,-52.591,173.523,18.784,153.240
C08650=1080.517,-120.360,-52.601,173.525,18.785,153.239
C08651=1080.523,-120.110,-52.611,173.527,18.786,153.239
C08652=1080.528,-119.860,-52.619,173.528,18.787,153.239
C08653=1080.534,-119.611,-52.629,173.529,18.787,153.239
C08654=1080.541,-119.361,-52.638,173.531,18.788,153.239
C08655=1080.547,-119.111,-52.647,173.533,18.789,153.239
C08656=1080.553,-118.862,-52.657,173.534,18.790,153.239
C08657=1080.560,-118.612,-52.666,173.536,18.791,153.239
C08658=1080.566,-118.362,-52.676,173.537,18.792,153.239
C08659=1080.571,-118.113,-52.685,173.539,18.793,153.238
C08660=1080.577,-117.862,-52.694,173.540,18.794,153.238
C08661=1080.583,-117.613,-52.703,173.542,18.795,153.238
C08662=1080.590,-117.363,-52.713,173.544,18.796,153.238
C08663=1080.596,-117.113,-52.723,173.545,18.796,153.238
C08664=1080.602,-116.863,-52.732,173.547,18.797,153.238
C08665=1080.608,-116.613,-52.742,173.548,18.798,153.238
C08666=1080.614,-116.364,-52.751,173.550,18.799,153.237
C08667=1080.621,-116.114,-52.760,173.552,18.800,153.237
C08668=1080.627,-115.865,-52.769,173.553,18.801,153.237
C08669=1080.633,-115.615,-52.779,173.554,18.801,153.237
C08670=1080.639,-115.365,-52.789,173.556,18.802,153.237
C08671=1080.645,-115.116,-52.798,173.558,18.803,153.237
C08672=1080.651,-114.866,-52.808,173.559,18.804,153.237
C08673=1080.658,-114.616,-52.817,173.561,18.805,153.237
C08674=1080.664,-114.366,-52.827,173.562,18.806,153.237
C08675=1080.670,-114.116,-52.836,173.563,18.807,153.237
C08676=1080.676,-113.840,-52.847,173.565,18.808,153.236
C08677=1080.683,-113.565,-52.857,173.567,18.809,153.236
C08678=1080.690,-113.288,-52.868,173.569,18.810,153.236
C08679=1080.697,-113.013,-52.879,173.570,18.811,153.236
C08680=1080.703,-112.763,-52.888,173.572,18.812,153.236
C08681=1080.709,-112.513,-52.898,173.574,18.813,153.236
C08682=1080.715,-112.263,-52.908,173.575,18.814,153.236
C08683=1080.721,-112.014,-52.917,173.577,18.815,153.236
C08684=1080.727,-111.765,-52.926,173.578,18.815,153.236
C08685=1080.733,-111.515,-52.936,173.579,18.817,153.236
C08686=1080.739,-111.265,-52.945,173.581,18.818,153.235
C08687=1080.745,-111.015,-52.955,173.583,18.819,153.235
C08688=1080.752,-110.765,-52.965,173.584,18.820,153.235
C08689=1080.757,-110.515,-52.975,173.586,18.821,153.235
C08690=1080.763,-110.266,-52.985,173.587,18.821,153.235
C08691=1080.770,-110.016,-52.995,173.589,18.822,153.235
C08692=1080.776,-109.766,-53.004,173.590,18.823,153.235
C08693=1080.782,-109.517,-53.014,173.592,18.824,153.235
C08694=1080.788,-109.267,-53.023,173.594,18.825,153.235
C08695=1080.794,-109.017,-53.033,173.595,18.826,153.234
C08696=1080.800,-108.767,-53.042,173.596,18.827,153.235
C08697=1080.807,-108.518,-53.052,173.598,18.828,153.234
C08698=1080.813,-108.268,-53.062,173.599,18.829,153.234
C08699=1080.819,-108.019,-53.072,173.601,18.830,153.234
C08700=1080.825,-107.768,-53.082,173.603,18.831,153.234
C08701=1080.831,-107.519,-53.092,173.604,18.832,153.234
C08702=1080.837,-107.269,-53.101,173.606,18.833,153.234
C08703=1080.843,-107.019,-53.111,173.607,18.834,153.234
C08704=1080.849,-106.769,-53.120,173.608,18.835,153.234
C08705=1080.856,-106.520,-53.131,173.610,18.836,153.234
C08706=1080.861,-106.270,-53.141,173.612,18.837,153.234
C08707=1080.867,-106.020,-53.150,173.614,18.838,153.233
C08708=1080.874,-105.770,-53.160,173.615,18.840,153.233
C08709=1080.880,-105.521,-53.169,173.617,18.841,153.233
C08710=1080.886,-105.271,-53.180,173.618,18.841,153.233
C08711=1080.892,-105.021,-53.190,173.619,18.842,153.233
C08712=1080.898,-104.771,-53.199,173.621,18.844,153.233
C08713=1080.904,-104.522,-53.209,173.622,18.845,153.233
C08714=1080.911,-104.272,-53.219,173.624,18.846,153.233
C08715=1080.916,-104.022,-53.229,173.626,18.847,153.233
C08716=1080.922,-103.773,-53.239,173.627,18.848,153.233
C08717=1080.928,-103.523,-53.249,173.629,18.849,153.233
C08718=1080.935,-103.274,-53.259,173.630,18.850,153.233
C08719=1080.940,-103.023,-53.269,173.631,18.851,153.233
C08720=1080.946,-102.774,-53.279,173.633,18.852,153.233
C08721=1080.953,-102.524,-53.288,173.635,18.853,153.232
C08722=1080.959,-102.275,-53.298,173.636,18.854,153.232
C08723=1080.964,-102.025,-53.309,173.638,18.856,153.232
C08724=1080.971,-101.775,-53.318,173.639,18.857,153.232
C08725=1080.977,-101.526,-53.328,173.641,18.858,153.232
C08726=1080.983,-101.276,-53.339,173.642,18.859,153.232
C08727=1080.989,-101.026,-53.348,173.643,18.860,153.232
C08728=1080.995,-100.777,-53.358,173.645,18.861,153.232
C08729=1081.001,-100.527,-53.368,173.647,18.862,153.232
C08730=1081.007,-100.277,-53.378,173.648,18.863,153.232
C08731=1081.013,-100.027,-53.388,173.650,18.864,153.232
C08732=1081.019,-99.778,-53.398,173.652,18.865,153.232
C08733=1081.025,-99.528,-53.408,173.653,18.867,153.232
C08734=1081.032,-99.278,-53.419,173.655,18.868,153.232
C08735=1081.038,-99.028,-53.428,173.656,18.868,153.232
C08736=1081.044,-98.778,-53.439,173.657,18.870,153.232
C08737=1081.050,-98.529,-53.449,173.659,18.871,153.231
C08738=1081.056,-98.279,-53.458,173.660,18.872,153.231
C08739=1081.062,-98.029,-53.469,173.662,18.873,153.231
C08740=1081.069,-97.750,-53.480,173.664,18.874,153.231
C08741=1081.076,-97.471,-53.492,173.665,18.876,153.231
C08742=1081.082,-97.192,-53.503,173.667,18.877,153.231
C08743=1081.089,-96.913,-53.514,173.668,18.878,153.231
C08744=1081.096,-96.664,-53.524,173.670,18.879,153.231
C08745=1081.101,-96.414,-53.534,173.671,18.881,153.231
C08746=1081.107,-96.164,-53.544,173.673,18.882,153.231
C08747=1081.113,-95.915,-53.555,173.674,18.883,153.231
C08748=1081.119,-95.665,-53.564,173.676,18.884,153.231
C08749=1081.125,-95.415,-53.575,173.678,18.886,153.231
C08750=1081.131,-95.166,-53.585,173.679,18.887,153.231
C08751=1081.137,-94.915,-53.596,173.681,18.888,153.231
C08752=1081.143,-94.665,-53.606,173.682,18.889,153.231
C08753=1081.149,-94.416,-53.617,173.684,18.891,153.231
C08754=1081.155,-94.166,-53.627,173.686,18.892,153.231
C08755=1081.161,-93.917,-53.637,173.686,18.893,153.231
C08756=1081.167,-93.667,-53.647,173.688,18.894,153.231
C08757=1081.173,-93.417,-53.657,173.689,18.895,153.231
C08758=1081.178,-93.167,-53.668,173.691,18.896,153.231
C08759=1081.185,-92.918,-53.678,173.692,18.898,153.231
C08760=1081.190,-92.668,-53.688,173.694,18.899,153.230
C08761=1081.197,-92.418,-53.699,173.696,18.900,153.230
C08762=1081.203,-92.168,-53.709,173.697,18.901,153.230
C08763=1081.209,-91.919,-53.719,173.699,18.903,153.230
C08764=1081.215,-91.669,-53.730,173.700,18.904,153.230
C08765=1081.221,-91.420,-53.740,173.702,18.905,153.230
C08766=1081.227,-91.170,-53.751,173.703,18.907,153.230
C08767=1081.232,-90.920,-53.761,173.705,18.908,153.230
C08768=1081.239,-90.671,-53.771,173.706,18.909,153.230
C08769=1081.245,-90.420,-53.781,173.707,18.910,153.230
C08770=1081.251,-90.171,-53.792,173.709,18.911,153.230
C08771=1081.257,-89.921,-53.803,173.711,18.912,153.230
C08772=1081.263,-89.672,-53.812,173.712,18.914,153.230
C08773=1081.269,-89.422,-53.823,173.713,18.916,153.230
C08774=1081.275,-89.172,-53.833,173.715,18.917,153.230
C08775=1081.282,-88.922,-53.844,173.717,18.918,153.230
C08776=1081.287,-88.673,-53.855,173.718,18.919,153.230
C08777=1081.294,-88.423,-53.864,173.720,18.921,153.230
C08778=1081.299,-88.173,-53.875,173.721,18.922,153.230
C08779=1081.306,-87.924,-53.885,173.723,18.923,153.230
C08780=1081.311,-87.674,-53.896,173.724,18.925,153.230
C08781=1081.318,-87.424,-53.907,173.726,18.926,153.230
C08782=1081.324,-87.175,-53.917,173.727,18.927,153.230
C08783=1081.329,-86.925,-53.927,173.729,18.929,153.230
C08784=1081.336,-86.675,-53.938,173.731,18.930,153.230
C08785=1081.342,-86.426,-53.949,173.732,18.931,153.230
C08786=1081.348,-86.176,-53.960,173.733,18.932,153.230
C08787=1081.354,-85.926,-53.969,173.734,18.933,153.230
C08788=1081.360,-85.676,-53.980,173.736,18.935,153.230
C08789=1081.366,-85.427,-53.990,173.737,18.936,153.230
C08790=1081.372,-85.176,-54.001,173.739,18.937,153.230
C08791=1081.378,-84.927,-54.012,173.740,18.939,153.230
C08792=1081.385,-84.678,-54.022,173.742,18.940,153.230
C08793=1081.390,-84.428,-54.033,173.743,18.941,153.230
C08794=1081.396,-84.177,-54.044,173.745,18.943,153.230
C08795=1081.403,-83.928,-54.054,173.747,18.944,153.230
C08796=1081.409,-83.679,-54.065,173.748,18.945,153.230
C08797=1081.415,-83.430,-54.075,173.750,18.947,153.230
C08798=1081.421,-83.179,-54.086,173.751,18.948,153.229
C08799=1081.427,-82.929,-54.096,173.753,18.949,153.230
C08800=1081.433,-82.680,-54.107,173.754,18.951,153.230
C08801=1081.439,-82.431,-54.118,173.756,18.952,153.230
C08802=1081.445,-82.180,-54.129,173.757,18.953,153.229
C08803=1081.452,-81.931,-54.139,173.759,18.955,153.229
C08804=1081.458,-81.654,-54.151,173.760,18.956,153.230
C08805=1081.465,-81.377,-54.162,173.762,18.957,153.229
C08806=1081.471,-81.100,-54.175,173.763,18.959,153.229
C08807=1081.479,-80.823,-54.186,173.766,18.961,153.229
C08808=1081.485,-80.574,-54.197,173.767,18.962,153.229
C08809=1081.491,-80.325,-54.208,173.769,18.963,153.229
C08810=1081.497,-80.075,-54.218,173.769,18.964,153.229
C08811=1081.503,-79.825,-54.230,173.771,18.966,153.229
C08812=1081.509,-79.576,-54.241,173.772,18.967,153.229
C08813=1081.515,-79.326,-54.250,173.774,18.969,153.230
C08814=1081.521,-79.076,-54.261,173.775,18.970,153.229
C08815=1081.527,-78.826,-54.272,173.777,18.972,153.229
C08816=1081.533,-78.577,-54.283,173.778,18.973,153.229
C08817=1081.539,-78.327,-54.294,173.780,18.975,153.229
C08818=1081.545,-78.077,-54.305,173.781,18.976,153.230
C08819=1081.551,-77.828,-54.316,173.783,18.977,153.229
C08820=1081.557,-77.578,-54.326,173.784,18.979,153.229
C08821=1081.563,-77.329,-54.337,173.786,18.980,153.229
C08822=1081.569,-77.079,-54.349,173.787,18.982,153.229
C08823=1081.575,-76.829,-54.359,173.789,18.983,153.230
C08824=1081.581,-76.580,-54.370,173.790,18.985,153.230
C08825=1081.587,-76.329,-54.382,173.792,18.986,153.230
C08826=1081.594,-76.080,-54.392,173.793,18.987,153.229
C08827=1081.599,-75.831,-54.403,173.795,18.989,153.229
C08828=1081.606,-75.581,-54.414,173.796,18.990,153.230
C08829=1081.611,-75.330,-54.424,173.798,18.992,153.230
C08830=1081.617,-75.081,-54.435,173.799,18.993,153.230
C08831=1081.623,-74.831,-54.447,173.801,18.995,153.230
C08832=1081.629,-74.582,-54.458,173.802,18.996,153.230
C08833=1081.635,-74.332,-54.469,173.803,18.998,153.230
C08834=1081.641,-74.082,-54.480,173.805,18.999,153.230
C08835=1081.647,-73.833,-54.491,173.807,19.000,153.230
C08836=1081.653,-73.583,-54.502,173.808,19.002,153.230
C08837=1081.658,-73.334,-54.513,173.809,19.003,153.230
C08838=1081.665,-73.084,-54.524,173.811,19.005,153.230
C08839=1081.671,-72.834,-54.535,173.812,19.006,153.230
C08840=1081.676,-72.585,-54.546,173.814,19.008,153.230
C08841=1081.683,-72.334,-54.557,173.815,19.009,153.230
C08842=1081.688,-72.085,-54.568,173.817,19.011,153.230
C08843=1081.694,-71.835,-54.579,173.818,19.013,153.230
C08844=1081.700,-71.585,-54.590,173.820,19.014,153.230
C08845=1081.706,-71.336,-54.601,173.822,19.016,153.230
C08846=1081.712,-71.086,-54.612,173.823,19.018,153.230
C08847=1081.717,-70.836,-54.623,173.825,19.019,153.230
C08848=1081.724,-70.587,-54.635,173.826,19.021,153.230
C08849=1081.729,-70.337,-54.646,173.828,19.022,153.230
C08850=1081.735,-70.088,-54.657,173.829,19.024,153.230
C08851=1081.741,-69.838,-54.668,173.830,19.026,153.230
C08852=1081.747,-69.588,-54.679,173.832,19.027,153.230
C08853=1081.753,-69.338,-54.690,173.833,19.029,153.230
C08854=1081.759,-69.089,-54.701,173.835,19.030,153.230
C08855=1081.765,-68.840,-54.713,173.836,19.032,153.230
C08856=1081.771,-68.589,-54.724,173.838,19.033,153.230
C08857=1081.777,-68.340,-54.735,173.839,19.035,153.230
C08858=1081.782,-68.090,-54.746,173.841,19.036,153.230
C08859=1081.789,-67.840,-54.757,173.842,19.038,153.230
C08860=1081.794,-67.591,-54.768,173.843,19.039,153.230
C08861=1081.800,-67.342,-54.780,173.845,19.041,153.230
C08862=1081.807,-67.091,-54.791,173.846,19.042,153.231
C08863=1081.812,-66.842,-54.803,173.848,19.044,153.231
C08864=1081.818,-66.591,-54.814,173.849,19.045,153.231
C08865=1081.824,-66.343,-54.825,173.851,19.047,153.231
C08866=1081.830,-66.093,-54.836,173.852,19.048,153.231
C08867=1081.836,-65.843,-54.848,173.854,19.050,153.231
C08868=1081.843,-65.569,-54.860,173.855,19.052,153.231
C08869=1081.849,-65.293,-54.873,173.857,19.054,153.231
C08870=1081.855,-65.020,-54.885,173.859,19.056,153.231
C08871=1081.862,-64.745,-54.897,173.860,19.057,153.231
C08872=1081.869,-64.495,-54.909,173.861,19.059,153.231
C08873=1081.874,-64.245,-54.920,173.863,19.060,153.231
C08874=1081.880,-63.995,-54.931,173.864,19.062,153.231
C08875=1081.886,-63.746,-54.943,173.866,19.064,153.231
C08876=1081.892,-63.496,-54.954,173.867,19.065,153.231
C08877=1081.898,-63.247,-54.965,173.869,19.067,153.231
C08878=1081.904,-62.998,-54.977,173.871,19.069,153.231
C08879=1081.910,-62.747,-54.989,173.872,19.070,153.231
C08880=1081.915,-62.498,-54.999,173.874,19.072,153.231
C08881=1081.922,-62.248,-55.011,173.875,19.073,153.231
C08882=1081.928,-61.999,-55.022,173.877,19.075,153.231
C08883=1081.934,-61.749,-55.033,173.878,19.076,153.231
C08884=1081.939,-61.499,-55.046,173.879,19.078,153.232
C08885=1081.946,-61.249,-55.057,173.881,19.080,153.232
C08886=1081.952,-61.000,-55.068,173.882,19.081,153.232
C08887=1081.958,-60.750,-55.080,173.884,19.083,153.232
C08888=1081.964,-60.501,-55.091,173.885,19.084,153.232
C08889=1081.970,-60.251,-55.103,173.887,19.086,153.232
C08890=1081.976,-60.001,-55.114,173.888,19.087,153.232
C08891=1081.982,-59.751,-55.125,173.889,19.090,153.232
C08892=1081.988,-59.502,-55.137,173.891,19.091,153.232
C08893=1081.994,-59.252,-55.149,173.892,19.093,153.232
C08894=1082.000,-59.003,-55.160,173.894,19.095,153.232
C08895=1082.006,-58.753,-55.172,173.896,19.096,153.232
C08896=1082.012,-58.504,-55.183,173.897,19.098,153.232
C08897=1082.018,-58.253,-55.195,173.899,19.099,153.232
C08898=1082.024,-58.004,-55.207,173.900,19.101,153.232
C08899=1082.030,-57.754,-55.218,173.901,19.103,153.232
C08900=1082.037,-57.505,-55.230,173.903,19.104,153.232
C08901=1082.042,-57.255,-55.241,173.904,19.106,153.232
C08902=1082.048,-57.005,-55.253,173.906,19.107,153.232
C08903=1082.054,-56.756,-55.264,173.907,19.109,153.232
C08904=1082.061,-56.506,-55.276,173.908,19.111,153.233
C08905=1082.066,-56.256,-55.288,173.910,19.112,153.233
C08906=1082.072,-56.007,-55.300,173.911,19.114,153.233
C08907=1082.079,-55.757,-55.311,173.913,19.115,153.233
C08908=1082.085,-55.508,-55.322,173.915,19.117,153.233
C08909=1082.090,-55.257,-55.334,173.917,19.119,153.233
C08910=1082.096,-55.008,-55.346,173.918,19.121,153.233
C08911=1082.103,-54.758,-55.357,173.919,19.122,153.233
C08912=1082.108,-54.509,-55.369,173.921,19.124,153.233
C08913=1082.114,-54.259,-55.380,173.922,19.125,153.233
C08914=1082.121,-54.009,-55.392,173.924,19.127,153.233
C08915=1082.127,-53.760,-55.404,173.925,19.129,153.233
C08916=1082.133,-53.510,-55.416,173.926,19.131,153.233
C08917=1082.139,-53.260,-55.428,173.928,19.132,153.233
C08918=1082.145,-53.011,-55.439,173.929,19.134,153.233
C08919=1082.151,-52.761,-55.451,173.931,19.135,153.233
C08920=1082.157,-52.512,-55.463,173.933,19.138,153.233
C08921=1082.163,-52.262,-55.474,173.934,19.139,153.233
C08922=1082.169,-52.012,-55.487,173.936,19.141,153.233
C08923=1082.175,-51.762,-55.497,173.937,19.142,153.233
C08924=1082.182,-51.513,-55.509,173.938,19.144,153.234
C08925=1082.188,-51.263,-55.522,173.940,19.146,153.234
C08926=1082.193,-51.014,-55.533,173.941,19.147,153.234
C08927=1082.200,-50.764,-55.545,173.943,19.149,153.234
C08928=1082.206,-50.514,-55.557,173.944,19.150,153.234
C08929=1082.212,-50.265,-55.568,173.945,19.152,153.234
C08930=1082.217,-50.015,-55.581,173.947,19.154,153.234
C08931=1082.224,-49.766,-55.592,173.949,19.156,153.234
C08932=1082.230,-49.492,-55.606,173.950,19.158,153.234
C08933=1082.237,-49.219,-55.619,173.952,19.159,153.234
C08934=1082.243,-48.945,-55.631,173.953,19.161,153.234
C08935=1082.250,-48.672,-55.644,173.955,19.163,153.234
C08936=1082.255,-48.422,-55.657,173.956,19.165,153.235
C08937=1082.261,-48.173,-55.669,173.958,19.167,153.235
C08938=1082.267,-47.923,-55.680,173.959,19.169,153.235
C08939=1082.272,-47.674,-55.693,173.961,19.171,153.235
C08940=1082.279,-47.424,-55.705,173.962,19.172,153.235
C08941=1082.285,-47.174,-55.717,173.963,19.174,153.235
C08942=1082.291,-46.925,-55.729,173.966,19.176,153.235
C08943=1082.297,-46.675,-55.741,173.967,19.178,153.235
C08944=1082.302,-46.425,-55.753,173.968,19.180,153.235
C08945=1082.309,-46.176,-55.765,173.970,19.181,153.235
C08946=1082.314,-45.926,-55.777,173.971,19.183,153.235
C08947=1082.319,-45.677,-55.789,173.972,19.185,153.235
C08948=1082.326,-45.427,-55.801,173.974,19.186,153.235
C08949=1082.332,-45.177,-55.813,173.975,19.188,153.236
C08950=1082.338,-44.928,-55.825,173.976,19.190,153.236
C08951=1082.344,-44.678,-55.837,173.979,19.192,153.236
C08952=1082.350,-44.428,-55.850,173.980,19.194,153.236
C08953=1082.356,-44.179,-55.861,173.981,19.195,153.236
C08954=1082.362,-43.929,-55.873,173.983,19.197,153.236
C08955=1082.367,-43.679,-55.886,173.984,19.199,153.236
C08956=1082.373,-43.430,-55.898,173.986,19.200,153.236
C08957=1082.379,-43.180,-55.910,173.987,19.202,153.236
C08958=1082.386,-42.931,-55.922,173.988,19.204,153.236
C08959=1082.392,-42.681,-55.935,173.990,19.207,153.236
C08960=1082.397,-42.432,-55.947,173.992,19.208,153.236
C08961=1082.404,-42.182,-55.958,173.993,19.210,153.236
C08962=1082.409,-41.932,-55.971,173.994,19.212,153.237
C08963=1082.415,-41.683,-55.983,173.996,19.213,153.237
C08964=1082.421,-41.433,-55.995,173.997,19.215,153.237
C08965=1082.427,-41.183,-56.007,173.999,19.217,153.237
C08966=1082.433,-40.933,-56.020,174.000,19.219,153.237
C08967=1082.439,-40.684,-56.031,174.002,19.221,153.237
C08968=1082.445,-40.434,-56.044,174.003,19.222,153.237
C08969=1082.451,-40.185,-56.057,174.005,19.224,153.237
C08970=1082.458,-39.935,-56.068,174.006,19.226,153.237
C08971=1082.463,-39.686,-56.081,174.007,19.228,153.237
C08972=1082.469,-39.436,-56.093,174.009,19.229,153.238
C08973=1082.475,-39.186,-56.106,174.010,19.231,153.238
C08974=1082.482,-38.936,-56.118,174.012,19.233,153.238
C08975=1082.487,-38.687,-56.130,174.014,19.235,153.238
C08976=1082.493,-38.437,-56.142,174.015,19.237,153.238
C08977=1082.499,-38.188,-56.155,174.016,19.238,153.238
C08978=1082.505,-37.938,-56.167,174.018,19.240,153.238
C08979=1082.511,-37.689,-56.179,174.019,19.242,153.238
C08980=1082.517,-37.439,-56.192,174.020,19.244,153.238
C08981=1082.522,-37.189,-56.204,174.023,19.246,153.238
C08982=1082.528,-36.940,-56.216,174.024,19.248,153.238
C08983=1082.534,-36.690,-56.229,174.025,19.250,153.239
C08984=1082.540,-36.440,-56.242,174.027,19.252,153.239
C08985=1082.546,-36.190,-56.254,174.028,19.254,153.239
C08986=1082.552,-35.941,-56.266,174.029,19.255,153.239
C08987=1082.557,-35.691,-56.278,174.030,19.257,153.239
C08988=1082.563,-35.442,-56.291,174.033,19.259,153.239
C08989=1082.569,-35.192,-56.303,174.034,19.261,153.239
C08990=1082.575,-34.943,-56.316,174.035,19.263,153.239
C08991=1082.581,-34.693,-56.329,174.037,19.265,153.239
C08992=1082.587,-34.443,-56.341,174.038,19.266,153.239
C08993=1082.593,-34.193,-56.354,174.039,19.268,153.240
C08994=1082.599,-33.944,-56.366,174.042,19.270,153.240
C08995=1082.605,-33.695,-56.378,174.043,19.272,153.240
C08996=1082.611,-33.422,-56.392,174.044,19.274,153.240
C08997=1082.618,-33.148,-56.406,174.046,19.276,153.240
C08998=1082.624,-32.876,-56.420,174.048,19.278,153.240
C08999=1082.630,-32.602,-56.433,174.049,19.280,153.240
C09000=1082.637,-32.353,-56.446,174.050,19.282,153.240
C09001=1082.642,-32.104,-56.458,174.052,19.284,153.241
C09002=1082.648,-31.854,-56.471,174.054,19.286,153.241
C09003=1082.654,-31.604,-56.483,174.055,19.288,153.241
C09004=1082.660,-31.355,-56.496,174.056,19.290,153.241
C09005=1082.666,-31.105,-56.509,174.058,19.292,153.241
C09006=1082.672,-30.855,-56.522,174.059,19.294,153.241
C09007=1082.677,-30.606,-56.534,174.060,19.295,153.241
C09008=1082.683,-30.356,-56.547,174.062,19.298,153.241
C09009=1082.689,-30.107,-56.560,174.064,19.299,153.241
C09010=1082.695,-29.857,-56.572,174.065,19.301,153.241
C09011=1082.701,-29.607,-56.585,174.067,19.303,153.242
C09012=1082.707,-29.357,-56.597,174.068,19.305,153.242
C09013=1082.713,-29.108,-56.611,174.069,19.306,153.242
C09014=1082.719,-28.858,-56.623,174.071,19.309,153.242
C09015=1082.725,-28.609,-56.635,174.073,19.311,153.242
C09016=1082.731,-28.360,-56.649,174.074,19.312,153.242
C09017=1082.737,-28.110,-56.661,174.075,19.314,153.242
C09018=1082.743,-27.860,-56.673,174.077,19.316,153.242
C09019=1082.749,-27.611,-56.686,174.078,19.318,153.242
C09020=1082.756,-27.361,-56.699,174.080,19.320,153.242
C09021=1082.761,-27.111,-56.712,174.081,19.322,153.243
C09022=1082.767,-26.861,-56.724,174.083,19.323,153.243
C09023=1082.773,-26.612,-56.738,174.084,19.325,153.243
C09024=1082.778,-26.363,-56.750,174.085,19.328,153.243
C09025=1082.784,-26.113,-56.763,174.087,19.329,153.243
C09026=1082.790,-25.864,-56.776,174.089,19.332,153.243
C09027=1082.796,-25.614,-56.789,174.090,19.334,153.243
C09028=1082.802,-25.364,-56.802,174.092,19.335,153.243
C09029=1082.808,-25.115,-56.814,174.093,19.337,153.244
C09030=1082.813,-24.864,-56.828,174.094,19.339,153.244
C09031=1082.819,-24.616,-56.840,174.096,19.341,153.244
C09032=1082.825,-24.366,-56.853,174.098,19.343,153.244
C09033=1082.831,-24.117,-56.866,174.099,19.345,153.244
C09034=1082.837,-23.867,-56.879,174.100,19.347,153.244
C09035=1082.843,-23.617,-56.891,174.101,19.349,153.244
C09036=1082.848,-23.367,-56.905,174.104,19.351,153.244
C09037=1082.854,-23.117,-56.918,174.105,19.353,153.244
C09038=1082.861,-22.868,-56.931,174.106,19.355,153.245
C09039=1082.867,-22.618,-56.944,174.107,19.357,153.245
C09040=1082.873,-22.369,-56.957,174.109,19.358,153.245
C09041=1082.878,-22.119,-56.970,174.110,19.360,153.245
C09042=1082.884,-21.870,-56.983,174.112,19.363,153.245
C09043=1082.889,-21.620,-56.996,174.114,19.364,153.245
C09044=1082.896,-21.371,-57.009,174.115,19.366,153.245
C09045=1082.902,-21.121,-57.021,174.116,19.368,153.246
C09046=1082.907,-20.872,-57.035,174.118,19.370,153.246
C09047=1082.913,-20.622,-57.048,174.120,19.373,153.246
C09048=1082.919,-20.373,-57.061,174.121,19.375,153.246
C09049=1082.925,-20.123,-57.074,174.122,19.376,153.246
C09050=1082.931,-19.873,-57.087,174.124,19.378,153.246
C09051=1082.936,-19.623,-57.100,174.125,19.380,153.246
C09052=1082.943,-19.374,-57.113,174.127,19.382,153.246
C09053=1082.949,-19.124,-57.126,174.128,19.384,153.246
C09054=1082.955,-18.875,-57.139,174.130,19.386,153.247
C09055=1082.960,-18.625,-57.153,174.131,19.388,153.247
C09056=1082.966,-18.375,-57.166,174.132,19.390,153.247
C09057=1082.972,-18.126,-57.179,174.134,19.392,153.247
C09058=1082.978,-17.876,-57.191,174.136,19.394,153.247
C09059=1082.985,-17.627,-57.205,174.137,19.396,153.247
C09060=1082.991,-17.353,-57.220,174.138,19.398,153.247
C09061=1082.997,-17.079,-57.234,174.140,19.400,153.247
C09062=1083.004,-16.806,-57.248,174.142,19.402,153.248
C09063=1083.010,-16.532,-57.262,174.144,19.404,153.248
C09064=1083.016,-16.282,-57.276,174.145,19.406,153.248
C09065=1083.022,-16.033,-57.289,174.146,19.408,153.248
C09066=1083.028,-15.783,-57.302,174.148,19.410,153.248
C09067=1083.034,-15.534,-57.315,174.150,19.412,153.248
C09068=1083.040,-15.284,-57.329,174.151,19.414,153.248
C09069=1083.045,-15.034,-57.342,174.152,19.416,153.248
C09070=1083.052,-14.785,-57.355,174.154,19.418,153.249
C09071=1083.057,-14.536,-57.369,174.155,19.420,153.249
C09072=1083.063,-14.286,-57.381,174.157,19.423,153.249
C09073=1083.069,-14.036,-57.395,174.158,19.424,153.249
C09074=1083.075,-13.787,-57.408,174.160,19.426,153.249
C09075=1083.080,-13.537,-57.422,174.161,19.428,153.249
C09076=1083.086,-13.287,-57.435,174.162,19.430,153.249
C09077=1083.092,-13.038,-57.448,174.164,19.432,153.249
C09078=1083.098,-12.789,-57.462,174.166,19.434,153.250
C09079=1083.104,-12.539,-57.475,174.167,19.436,153.250
C09080=1083.109,-12.289,-57.488,174.168,19.438,153.250
C09081=1083.115,-12.040,-57.502,174.170,19.440,153.250
C09082=1083.121,-11.790,-57.516,174.172,19.442,153.250
C09083=1083.127,-11.541,-57.529,174.173,19.444,153.250
C09084=1083.132,-11.291,-57.542,174.174,19.446,153.250
C09085=1083.138,-11.041,-57.555,174.176,19.448,153.251
C09086=1083.145,-10.791,-57.569,174.178,19.450,153.251
C09087=1083.151,-10.542,-57.583,174.179,19.452,153.251
C09088=1083.156,-10.292,-57.597,174.180,19.454,153.251
C09089=1083.162,-10.042,-57.609,174.182,19.456,153.251
C09090=1083.168,-9.793,-57.623,174.184,19.458,153.251
C09091=1083.174,-9.544,-57.636,174.185,19.460,153.251
C09092=1083.179,-9.294,-57.650,174.186,19.462,153.252
C09093=1083.186,-9.045,-57.663,174.188,19.464,153.252
